LIN {X -277.944,Y 0.000,Z 80.000,A 0.000,B 0.000,C 180.000,E1 0.000} C_DIS
LIN {X -277.576,Y -14.309,Z 80.000,A 0.000,B 0.000,C 180.000,E1 0.000} C_DIS
LIN {X -276.472,Y -28.580,Z 80.000,A 0.000,B 0.000,C 180.000,E1 0.000} C_DIS
LIN {X -274.635,Y -42.773,Z 80.000,A 0.000,B 0.000,C 180.000,E1 0.000} C_DIS
LIN {X -272.067,Y -56.854,Z 80.000,A 0.000,B 0.000,C 180.000,E1 0.000} C_DIS
LIN {X -268.780,Y -70.785,Z 80.000,A 0.000,B 0.000,C 180.000,E1 0.000} C_DIS
LIN {X -264.780,Y -84.527,Z 80.000,A 0.000,B 0.000,C 180.000,E1 0.000} C_DIS
LIN {X -260.078,Y -98.045,Z 80.000,A 0.000,B 0.000,C 180.000,E1 0.000} C_DIS
LIN {X -254.685,Y -111.305,Z 80.000,A 0.000,B 0.000,C 180.000,E1 0.000} C_DIS
LIN {X -248.618,Y -124.267,Z 80.000,A 0.000,B 0.000,C 180.000,E1 0.000} C_DIS
LIN {X -241.892,Y -136.901,Z 80.000,A 0.000,B 0.000,C 180.000,E1 0.000} C_DIS
LIN {X -234.523,Y -149.172,Z 80.000,A 0.000,B 0.000,C 180.000,E1 0.000} C_DIS
LIN {X -226.533,Y -161.047,Z 80.000,A 0.000,B 0.000,C 180.000,E1 0.000} C_DIS
LIN {X -217.943,Y -172.495,Z 80.000,A 0.000,B 0.000,C 180.000,E1 0.000} C_DIS
LIN {X -208.773,Y -183.486,Z 80.000,A 0.000,B 0.000,C 180.000,E1 0.000} C_DIS
LIN {X -199.051,Y -193.990,Z 80.000,A 0.000,B 0.000,C 180.000,E1 0.000} C_DIS
LIN {X -188.801,Y -203.979,Z 80.000,A 0.000,B 0.000,C 180.000,E1 0.000} C_DIS
LIN {X -178.050,Y -213.428,Z 80.000,A 0.000,B 0.000,C 180.000,E1 0.000} C_DIS
LIN {X -166.826,Y -222.311,Z 80.000,A 0.000,B 0.000,C 180.000,E1 0.000} C_DIS
LIN {X -155.161,Y -230.604,Z 80.000,A 0.000,B 0.000,C 180.000,E1 0.000} C_DIS
LIN {X -143.084,Y -238.286,Z 80.000,A 0.000,B 0.000,C 180.000,E1 0.000} C_DIS
LIN {X -130.627,Y -245.336,Z 80.000,A 0.000,B 0.000,C 180.000,E1 0.000} C_DIS
LIN {X -117.825,Y -251.735,Z 80.000,A 0.000,B 0.000,C 180.000,E1 0.000} C_DIS
LIN {X -104.709,Y -257.467,Z 80.000,A 0.000,B 0.000,C 180.000,E1 0.000} C_DIS
LIN {X -91.317,Y -262.516,Z 80.000,A 0.000,B 0.000,C 180.000,E1 0.000} C_DIS
LIN {X -77.682,Y -266.869,Z 80.000,A 0.000,B 0.000,C 180.000,E1 0.000} C_DIS
LIN {X -63.841,Y -270.513,Z 80.000,A 0.000,B 0.000,C 180.000,E1 0.000} C_DIS
LIN {X -49.830,Y -273.441,Z 80.000,A 0.000,B 0.000,C 180.000,E1 0.000} C_DIS
LIN {X -35.687,Y -275.644,Z 80.000,A 0.000,B 0.000,C 180.000,E1 0.000} C_DIS
LIN {X -21.451,Y -277.115,Z 80.000,A 0.000,B 0.000,C 180.000,E1 0.000} C_DIS
LIN {X -7.156,Y -277.853,Z 80.000,A 0.000,B 0.000,C 180.000,E1 0.000} C_DIS
LIN {X 7.156,Y -277.853,Z 80.000,A 0.000,B 0.000,C 180.000,E1 0.000} C_DIS
LIN {X 21.451,Y -277.115,Z 80.000,A 0.000,B 0.000,C 180.000,E1 0.000} C_DIS
LIN {X 35.687,Y -275.644,Z 80.000,A 0.000,B 0.000,C 180.000,E1 0.000} C_DIS
LIN {X 49.830,Y -273.441,Z 80.000,A 0.000,B 0.000,C 180.000,E1 0.000} C_DIS
LIN {X 63.841,Y -270.513,Z 80.000,A 0.000,B 0.000,C 180.000,E1 0.000} C_DIS
LIN {X 77.682,Y -266.869,Z 80.000,A 0.000,B 0.000,C 180.000,E1 0.000} C_DIS
LIN {X 91.317,Y -262.516,Z 80.000,A 0.000,B 0.000,C 180.000,E1 0.000} C_DIS
LIN {X 104.709,Y -257.467,Z 80.000,A 0.000,B 0.000,C 180.000,E1 0.000} C_DIS
LIN {X 117.825,Y -251.735,Z 80.000,A 0.000,B 0.000,C 180.000,E1 0.000} C_DIS
LIN {X 130.627,Y -245.336,Z 80.000,A 0.000,B 0.000,C 180.000,E1 0.000} C_DIS
LIN {X 143.084,Y -238.286,Z 80.000,A 0.000,B 0.000,C 180.000,E1 0.000} C_DIS
LIN {X 155.161,Y -230.604,Z 80.000,A 0.000,B 0.000,C 180.000,E1 0.000} C_DIS
LIN {X 166.826,Y -222.311,Z 80.000,A 0.000,B 0.000,C 180.000,E1 0.000} C_DIS
LIN {X 178.050,Y -213.428,Z 80.000,A 0.000,B 0.000,C 180.000,E1 0.000} C_DIS
LIN {X 188.801,Y -203.979,Z 80.000,A 0.000,B 0.000,C 180.000,E1 0.000} C_DIS
LIN {X 199.051,Y -193.990,Z 80.000,A 0.000,B 0.000,C 180.000,E1 0.000} C_DIS
LIN {X 208.773,Y -183.486,Z 80.000,A 0.000,B 0.000,C 180.000,E1 0.000} C_DIS
LIN {X 217.943,Y -172.495,Z 80.000,A 0.000,B 0.000,C 180.000,E1 0.000} C_DIS
LIN {X 226.533,Y -161.047,Z 80.000,A 0.000,B 0.000,C 180.000,E1 0.000} C_DIS
LIN {X 234.523,Y -149.172,Z 80.000,A 0.000,B 0.000,C 180.000,E1 0.000} C_DIS
LIN {X 241.892,Y -136.901,Z 80.000,A 0.000,B 0.000,C 180.000,E1 0.000} C_DIS
LIN {X 248.618,Y -124.268,Z 80.000,A 0.000,B 0.000,C 180.000,E1 0.000} C_DIS
LIN {X 254.686,Y -111.304,Z 80.000,A 0.000,B 0.000,C 180.000,E1 0.000} C_DIS
LIN {X 260.078,Y -98.045,Z 80.000,A 0.000,B 0.000,C 180.000,E1 0.000} C_DIS
LIN {X 264.780,Y -84.527,Z 80.000,A 0.000,B 0.000,C 180.000,E1 0.000} C_DIS
LIN {X 268.780,Y -70.785,Z 80.000,A 0.000,B 0.000,C 180.000,E1 0.000} C_DIS
LIN {X 272.067,Y -56.854,Z 80.000,A 0.000,B 0.000,C 180.000,E1 0.000} C_DIS
LIN {X 274.635,Y -42.773,Z 80.000,A 0.000,B 0.000,C 180.000,E1 0.000} C_DIS
LIN {X 276.472,Y -28.580,Z 80.000,A 0.000,B 0.000,C 180.000,E1 0.000} C_DIS
LIN {X 277.576,Y -14.309,Z 80.000,A 0.000,B 0.000,C 180.000,E1 0.000} C_DIS
LIN {X 277.944,Y 0.000,Z 80.000,A 0.000,B 0.000,C 180.000,E1 0.000} C_DIS
LIN {X 277.576,Y 14.309,Z 80.000,A 0.000,B 0.000,C 180.000,E1 0.000} C_DIS
LIN {X 276.472,Y 28.580,Z 80.000,A 0.000,B 0.000,C 180.000,E1 0.000} C_DIS
LIN {X 274.635,Y 42.773,Z 80.000,A 0.000,B 0.000,C 180.000,E1 0.000} C_DIS
LIN {X 272.067,Y 56.854,Z 80.000,A 0.000,B 0.000,C 180.000,E1 0.000} C_DIS
LIN {X 268.780,Y 70.785,Z 80.000,A 0.000,B 0.000,C 180.000,E1 0.000} C_DIS
LIN {X 264.780,Y 84.527,Z 80.000,A 0.000,B 0.000,C 180.000,E1 0.000} C_DIS
LIN {X 260.078,Y 98.045,Z 80.000,A 0.000,B 0.000,C 180.000,E1 0.000} C_DIS
LIN {X 254.685,Y 111.305,Z 80.000,A 0.000,B 0.000,C 180.000,E1 0.000} C_DIS
LIN {X 252.753,Y 115.434,Z 80.000,A 0.000,B 0.000,C 180.000,E1 0.000} C_DIS
LIN {X 248.618,Y 124.267,Z 80.000,A 0.000,B 0.000,C 180.000,E1 0.000} C_DIS
LIN {X 241.892,Y 136.901,Z 80.000,A 0.000,B 0.000,C 180.000,E1 0.000} C_DIS
LIN {X 234.523,Y 149.172,Z 80.000,A 0.000,B 0.000,C 180.000,E1 0.000} C_DIS
LIN {X 226.533,Y 161.047,Z 80.000,A 0.000,B 0.000,C 180.000,E1 0.000} C_DIS
LIN {X 217.943,Y 172.495,Z 80.000,A 0.000,B 0.000,C 180.000,E1 0.000} C_DIS
LIN {X 208.773,Y 183.486,Z 80.000,A 0.000,B 0.000,C 180.000,E1 0.000} C_DIS
LIN {X 199.051,Y 193.990,Z 80.000,A 0.000,B 0.000,C 180.000,E1 0.000} C_DIS
LIN {X 188.801,Y 203.979,Z 80.000,A 0.000,B 0.000,C 180.000,E1 0.000} C_DIS
LIN {X 178.050,Y 213.428,Z 80.000,A 0.000,B 0.000,C 180.000,E1 0.000} C_DIS
LIN {X 166.826,Y 222.311,Z 80.000,A 0.000,B 0.000,C 180.000,E1 0.000} C_DIS
LIN {X 155.161,Y 230.604,Z 80.000,A 0.000,B 0.000,C 180.000,E1 0.000} C_DIS
LIN {X 143.084,Y 238.286,Z 80.000,A 0.000,B 0.000,C 180.000,E1 0.000} C_DIS
LIN {X 130.627,Y 245.336,Z 80.000,A 0.000,B 0.000,C 180.000,E1 0.000} C_DIS
LIN {X 117.825,Y 251.735,Z 80.000,A 0.000,B 0.000,C 180.000,E1 0.000} C_DIS
LIN {X 104.709,Y 257.467,Z 80.000,A 0.000,B 0.000,C 180.000,E1 0.000} C_DIS
LIN {X 91.317,Y 262.516,Z 80.000,A 0.000,B 0.000,C 180.000,E1 0.000} C_DIS
LIN {X 77.682,Y 266.869,Z 80.000,A 0.000,B 0.000,C 180.000,E1 0.000} C_DIS
;rapid-leaky
$VEL.CP=0.3
LIN {X 73.337,Y 251.943,Z 80.000,A 0.000,B 0.000,C 180.000,E1 0.000} C_DIS
;bead-perimeter_inner
$VEL.CP=0.73
LIN {X 60.270,Y 255.384,Z 80.000,A 0.000,B 0.000,C 180.000,E1 0.000} C_DIS
LIN {X 47.043,Y 258.148,Z 80.000,A 0.000,B 0.000,C 180.000,E1 0.000} C_DIS
LIN {X 33.691,Y 260.228,Z 80.000,A 0.000,B 0.000,C 180.000,E1 0.000} C_DIS
LIN {X 20.251,Y 261.617,Z 80.000,A 0.000,B 0.000,C 180.000,E1 0.000} C_DIS
LIN {X 6.755,Y 262.313,Z 80.000,A 0.000,B 0.000,C 180.000,E1 0.000} C_DIS
LIN {X -6.755,Y 262.313,Z 80.000,A 0.000,B 0.000,C 180.000,E1 0.000} C_DIS
LIN {X -20.251,Y 261.617,Z 80.000,A 0.000,B 0.000,C 180.000,E1 0.000} C_DIS
LIN {X -33.691,Y 260.228,Z 80.000,A 0.000,B 0.000,C 180.000,E1 0.000} C_DIS
LIN {X -47.043,Y 258.148,Z 80.000,A 0.000,B 0.000,C 180.000,E1 0.000} C_DIS
LIN {X -60.270,Y 255.384,Z 80.000,A 0.000,B 0.000,C 180.000,E1 0.000} C_DIS
LIN {X -73.337,Y 251.943,Z 80.000,A 0.000,B 0.000,C 180.000,E1 0.000} C_DIS
LIN {X -86.210,Y 247.833,Z 80.000,A 0.000,B 0.000,C 180.000,E1 0.000} C_DIS
LIN {X -98.853,Y 243.067,Z 80.000,A 0.000,B 0.000,C 180.000,E1 0.000} C_DIS
LIN {X -111.235,Y 237.656,Z 80.000,A 0.000,B 0.000,C 180.000,E1 0.000} C_DIS
LIN {X -123.321,Y 231.615,Z 80.000,A 0.000,B 0.000,C 180.000,E1 0.000} C_DIS
LIN {X -135.081,Y 224.959,Z 80.000,A 0.000,B 0.000,C 180.000,E1 0.000} C_DIS
LIN {X -146.484,Y 217.706,Z 80.000,A 0.000,B 0.000,C 180.000,E1 0.000} C_DIS
LIN {X -157.496,Y 209.877,Z 80.000,A 0.000,B 0.000,C 180.000,E1 0.000} C_DIS
LIN {X -168.092,Y 201.491,Z 80.000,A 0.000,B 0.000,C 180.000,E1 0.000} C_DIS
LIN {X -178.242,Y 192.570,Z 80.000,A 0.000,B 0.000,C 180.000,E1 0.000} C_DIS
LIN {X -187.918,Y 183.141,Z 80.000,A 0.000,B 0.000,C 180.000,E1 0.000} C_DIS
LIN {X -197.096,Y 173.224,Z 80.000,A 0.000,B 0.000,C 180.000,E1 0.000} C_DIS
LIN {X -205.754,Y 162.847,Z 80.000,A 0.000,B 0.000,C 180.000,E1 0.000} C_DIS
LIN {X -213.863,Y 152.040,Z 80.000,A 0.000,B 0.000,C 180.000,E1 0.000} C_DIS
LIN {X -221.406,Y 140.829,Z 80.000,A 0.000,B 0.000,C 180.000,E1 0.000} C_DIS
LIN {X -228.363,Y 129.244,Z 80.000,A 0.000,B 0.000,C 180.000,E1 0.000} C_DIS
LIN {X -234.713,Y 117.317,Z 80.000,A 0.000,B 0.000,C 180.000,E1 0.000} C_DIS
LIN {X -240.441,Y 105.079,Z 80.000,A 0.000,B 0.000,C 180.000,E1 0.000} C_DIS
LIN {X -245.532,Y 92.562,Z 80.000,A 0.000,B 0.000,C 180.000,E1 0.000} C_DIS
LIN {X -249.971,Y 79.800,Z 80.000,A 0.000,B 0.000,C 180.000,E1 0.000} C_DIS
LIN {X -253.748,Y 66.826,Z 80.000,A 0.000,B 0.000,C 180.000,E1 0.000} C_DIS
LIN {X -256.851,Y 53.674,Z 80.000,A 0.000,B 0.000,C 180.000,E1 0.000} C_DIS
LIN {X -259.275,Y 40.380,Z 80.000,A 0.000,B 0.000,C 180.000,E1 0.000} C_DIS
LIN {X -261.009,Y 26.982,Z 80.000,A 0.000,B 0.000,C 180.000,E1 0.000} C_DIS
LIN {X -262.051,Y 13.509,Z 80.000,A 0.000,B 0.000,C 180.000,E1 0.000} C_DIS
LIN {X -262.399,Y 0.000,Z 80.000,A 0.000,B 0.000,C 180.000,E1 0.000} C_DIS
LIN {X -262.051,Y -13.509,Z 80.000,A 0.000,B 0.000,C 180.000,E1 0.000} C_DIS
LIN {X -261.009,Y -26.982,Z 80.000,A 0.000,B 0.000,C 180.000,E1 0.000} C_DIS
LIN {X -259.275,Y -40.380,Z 80.000,A 0.000,B 0.000,C 180.000,E1 0.000} C_DIS
LIN {X -256.851,Y -53.674,Z 80.000,A 0.000,B 0.000,C 180.000,E1 0.000} C_DIS
LIN {X -253.748,Y -66.826,Z 80.000,A 0.000,B 0.000,C 180.000,E1 0.000} C_DIS
LIN {X -249.971,Y -79.800,Z 80.000,A 0.000,B 0.000,C 180.000,E1 0.000} C_DIS
LIN {X -245.532,Y -92.562,Z 80.000,A 0.000,B 0.000,C 180.000,E1 0.000} C_DIS
LIN {X -240.441,Y -105.080,Z 80.000,A 0.000,B 0.000,C 180.000,E1 0.000} C_DIS
LIN {X -234.713,Y -117.317,Z 80.000,A 0.000,B 0.000,C 180.000,E1 0.000} C_DIS
LIN {X -228.363,Y -129.244,Z 80.000,A 0.000,B 0.000,C 180.000,E1 0.000} C_DIS
LIN {X -221.406,Y -140.829,Z 80.000,A 0.000,B 0.000,C 180.000,E1 0.000} C_DIS
LIN {X -213.863,Y -152.040,Z 80.000,A 0.000,B 0.000,C 180.000,E1 0.000} C_DIS
LIN {X -205.754,Y -162.847,Z 80.000,A 0.000,B 0.000,C 180.000,E1 0.000} C_DIS
LIN {X -197.096,Y -173.224,Z 80.000,A 0.000,B 0.000,C 180.000,E1 0.000} C_DIS
LIN {X -187.918,Y -183.141,Z 80.000,A 0.000,B 0.000,C 180.000,E1 0.000} C_DIS
LIN {X -178.242,Y -192.570,Z 80.000,A 0.000,B 0.000,C 180.000,E1 0.000} C_DIS
LIN {X -168.092,Y -201.491,Z 80.000,A 0.000,B 0.000,C 180.000,E1 0.000} C_DIS
LIN {X -157.496,Y -209.877,Z 80.000,A 0.000,B 0.000,C 180.000,E1 0.000} C_DIS
LIN {X -146.484,Y -217.706,Z 80.000,A 0.000,B 0.000,C 180.000,E1 0.000} C_DIS
LIN {X -135.081,Y -224.959,Z 80.000,A 0.000,B 0.000,C 180.000,E1 0.000} C_DIS
LIN {X -123.321,Y -231.615,Z 80.000,A 0.000,B 0.000,C 180.000,E1 0.000} C_DIS
LIN {X -111.235,Y -237.656,Z 80.000,A 0.000,B 0.000,C 180.000,E1 0.000} C_DIS
LIN {X -98.853,Y -243.067,Z 80.000,A 0.000,B 0.000,C 180.000,E1 0.000} C_DIS
LIN {X -86.210,Y -247.833,Z 80.000,A 0.000,B 0.000,C 180.000,E1 0.000} C_DIS
LIN {X -73.337,Y -251.943,Z 80.000,A 0.000,B 0.000,C 180.000,E1 0.000} C_DIS
LIN {X -60.270,Y -255.384,Z 80.000,A 0.000,B 0.000,C 180.000,E1 0.000} C_DIS
LIN {X -47.043,Y -258.148,Z 80.000,A 0.000,B 0.000,C 180.000,E1 0.000} C_DIS
LIN {X -33.691,Y -260.228,Z 80.000,A 0.000,B 0.000,C 180.000,E1 0.000} C_DIS
LIN {X -20.251,Y -261.617,Z 80.000,A 0.000,B 0.000,C 180.000,E1 0.000} C_DIS
LIN {X -6.755,Y -262.313,Z 80.000,A 0.000,B 0.000,C 180.000,E1 0.000} C_DIS
LIN {X 6.755,Y -262.313,Z 80.000,A 0.000,B 0.000,C 180.000,E1 0.000} C_DIS
LIN {X 20.251,Y -261.617,Z 80.000,A 0.000,B 0.000,C 180.000,E1 0.000} C_DIS
LIN {X 33.691,Y -260.228,Z 80.000,A 0.000,B 0.000,C 180.000,E1 0.000} C_DIS
LIN {X 47.043,Y -258.148,Z 80.000,A 0.000,B 0.000,C 180.000,E1 0.000} C_DIS
LIN {X 60.270,Y -255.384,Z 80.000,A 0.000,B 0.000,C 180.000,E1 0.000} C_DIS
LIN {X 73.337,Y -251.943,Z 80.000,A 0.000,B 0.000,C 180.000,E1 0.000} C_DIS
LIN {X 86.210,Y -247.833,Z 80.000,A 0.000,B 0.000,C 180.000,E1 0.000} C_DIS
LIN {X 98.853,Y -243.067,Z 80.000,A 0.000,B 0.000,C 180.000,E1 0.000} C_DIS
LIN {X 111.235,Y -237.656,Z 80.000,A 0.000,B 0.000,C 180.000,E1 0.000} C_DIS
LIN {X 123.321,Y -231.615,Z 80.000,A 0.000,B 0.000,C 180.000,E1 0.000} C_DIS
LIN {X 135.081,Y -224.959,Z 80.000,A 0.000,B 0.000,C 180.000,E1 0.000} C_DIS
LIN {X 146.484,Y -217.706,Z 80.000,A 0.000,B 0.000,C 180.000,E1 0.000} C_DIS
LIN {X 157.496,Y -209.877,Z 80.000,A 0.000,B 0.000,C 180.000,E1 0.000} C_DIS
LIN {X 168.092,Y -201.491,Z 80.000,A 0.000,B 0.000,C 180.000,E1 0.000} C_DIS
LIN {X 178.242,Y -192.570,Z 80.000,A 0.000,B 0.000,C 180.000,E1 0.000} C_DIS
LIN {X 187.918,Y -183.141,Z 80.000,A 0.000,B 0.000,C 180.000,E1 0.000} C_DIS
LIN {X 197.096,Y -173.224,Z 80.000,A 0.000,B 0.000,C 180.000,E1 0.000} C_DIS
LIN {X 205.754,Y -162.847,Z 80.000,A 0.000,B 0.000,C 180.000,E1 0.000} C_DIS
LIN {X 213.863,Y -152.040,Z 80.000,A 0.000,B 0.000,C 180.000,E1 0.000} C_DIS
LIN {X 221.406,Y -140.829,Z 80.000,A 0.000,B 0.000,C 180.000,E1 0.000} C_DIS
LIN {X 228.363,Y -129.244,Z 80.000,A 0.000,B 0.000,C 180.000,E1 0.000} C_DIS
LIN {X 234.713,Y -117.317,Z 80.000,A 0.000,B 0.000,C 180.000,E1 0.000} C_DIS
LIN {X 240.441,Y -105.079,Z 80.000,A 0.000,B 0.000,C 180.000,E1 0.000} C_DIS
LIN {X 245.532,Y -92.562,Z 80.000,A 0.000,B 0.000,C 180.000,E1 0.000} C_DIS
LIN {X 249.971,Y -79.800,Z 80.000,A 0.000,B 0.000,C 180.000,E1 0.000} C_DIS
LIN {X 253.748,Y -66.826,Z 80.000,A 0.000,B 0.000,C 180.000,E1 0.000} C_DIS
LIN {X 256.851,Y -53.674,Z 80.000,A 0.000,B 0.000,C 180.000,E1 0.000} C_DIS
LIN {X 259.275,Y -40.380,Z 80.000,A 0.000,B 0.000,C 180.000,E1 0.000} C_DIS
LIN {X 261.009,Y -26.982,Z 80.000,A 0.000,B 0.000,C 180.000,E1 0.000} C_DIS
LIN {X 262.051,Y -13.509,Z 80.000,A 0.000,B 0.000,C 180.000,E1 0.000} C_DIS
LIN {X 262.399,Y 0.000,Z 80.000,A 0.000,B 0.000,C 180.000,E1 0.000} C_DIS
LIN {X 262.051,Y 13.509,Z 80.000,A 0.000,B 0.000,C 180.000,E1 0.000} C_DIS
LIN {X 261.009,Y 26.982,Z 80.000,A 0.000,B 0.000,C 180.000,E1 0.000} C_DIS
LIN {X 259.275,Y 40.380,Z 80.000,A 0.000,B 0.000,C 180.000,E1 0.000} C_DIS
LIN {X 256.851,Y 53.674,Z 80.000,A 0.000,B 0.000,C 180.000,E1 0.000} C_DIS
LIN {X 253.748,Y 66.826,Z 80.000,A 0.000,B 0.000,C 180.000,E1 0.000} C_DIS
LIN {X 249.971,Y 79.800,Z 80.000,A 0.000,B 0.000,C 180.000,E1 0.000} C_DIS
LIN {X 245.532,Y 92.562,Z 80.000,A 0.000,B 0.000,C 180.000,E1 0.000} C_DIS
LIN {X 240.441,Y 105.080,Z 80.000,A 0.000,B 0.000,C 180.000,E1 0.000} C_DIS
LIN {X 238.678,Y 108.847,Z 80.000,A 0.000,B 0.000,C 180.000,E1 0.000} C_DIS
LIN {X 234.713,Y 117.317,Z 80.000,A 0.000,B 0.000,C 180.000,E1 0.000} C_DIS
LIN {X 228.363,Y 129.244,Z 80.000,A 0.000,B 0.000,C 180.000,E1 0.000} C_DIS
LIN {X 221.406,Y 140.829,Z 80.000,A 0.000,B 0.000,C 180.000,E1 0.000} C_DIS
LIN {X 213.863,Y 152.040,Z 80.000,A 0.000,B 0.000,C 180.000,E1 0.000} C_DIS
LIN {X 205.754,Y 162.847,Z 80.000,A 0.000,B 0.000,C 180.000,E1 0.000} C_DIS
LIN {X 197.096,Y 173.224,Z 80.000,A 0.000,B 0.000,C 180.000,E1 0.000} C_DIS
LIN {X 187.918,Y 183.141,Z 80.000,A 0.000,B 0.000,C 180.000,E1 0.000} C_DIS
LIN {X 178.242,Y 192.570,Z 80.000,A 0.000,B 0.000,C 180.000,E1 0.000} C_DIS
LIN {X 168.092,Y 201.491,Z 80.000,A 0.000,B 0.000,C 180.000,E1 0.000} C_DIS
LIN {X 157.496,Y 209.877,Z 80.000,A 0.000,B 0.000,C 180.000,E1 0.000} C_DIS
LIN {X 146.484,Y 217.706,Z 80.000,A 0.000,B 0.000,C 180.000,E1 0.000} C_DIS
LIN {X 135.081,Y 224.959,Z 80.000,A 0.000,B 0.000,C 180.000,E1 0.000} C_DIS
LIN {X 123.321,Y 231.615,Z 80.000,A 0.000,B 0.000,C 180.000,E1 0.000} C_DIS
LIN {X 111.235,Y 237.656,Z 80.000,A 0.000,B 0.000,C 180.000,E1 0.000} C_DIS
LIN {X 98.853,Y 243.067,Z 80.000,A 0.000,B 0.000,C 180.000,E1 0.000} C_DIS
LIN {X 86.210,Y 247.833,Z 80.000,A 0.000,B 0.000,C 180.000,E1 0.000} C_DIS
LIN {X 73.337,Y 251.943,Z 80.000,A 0.000,B 0.000,C 180.000,E1 0.000} C_DIS
;rapid-leaky
$VEL.CP=0.3
LIN {X -163.493,Y 181.889,Z 80.000,A 0.000,B 0.000,C 180.000,E1 0.000} C_DIS
;bead-sparse_infill
$VEL.CP=0.73
LIN {X -182.087,Y 163.294,Z 80.000,A 0.000,B 0.000,C 180.000,E1 0.000} C_DIS
LIN {X -183.751,Y 161.496,Z 80.000,A 0.000,B 0.000,C 180.000,E1 0.000} C_DIS
LIN {X -191.823,Y 151.821,Z 80.000,A 0.000,B 0.000,C 180.000,E1 0.000} C_DIS
LIN {X -199.383,Y 141.747,Z 80.000,A 0.000,B 0.000,C 180.000,E1 0.000} C_DIS
LIN {X -206.416,Y 131.294,Z 80.000,A 0.000,B 0.000,C 180.000,E1 0.000} C_DIS
LIN {X -212.902,Y 120.493,Z 80.000,A 0.000,B 0.000,C 180.000,E1 0.000} C_DIS
LIN {X -218.822,Y 109.374,Z 80.000,A 0.000,B 0.000,C 180.000,E1 0.000} C_DIS
LIN {X -224.162,Y 97.965,Z 80.000,A 0.000,B 0.000,C 180.000,E1 0.000} C_DIS
LIN {X -228.908,Y 86.295,Z 80.000,A 0.000,B 0.000,C 180.000,E1 0.000} C_DIS
LIN {X -233.047,Y 74.397,Z 80.000,A 0.000,B 0.000,C 180.000,E1 0.000} C_DIS
LIN {X -236.567,Y 62.302,Z 80.000,A 0.000,B 0.000,C 180.000,E1 0.000} C_DIS
LIN {X -239.461,Y 50.040,Z 80.000,A 0.000,B 0.000,C 180.000,E1 0.000} C_DIS
LIN {X -241.721,Y 37.645,Z 80.000,A 0.000,B 0.000,C 180.000,E1 0.000} C_DIS
LIN {X -243.338,Y 25.156,Z 80.000,A 0.000,B 0.000,C 180.000,E1 0.000} C_DIS
LIN {X -244.309,Y 12.595,Z 80.000,A 0.000,B 0.000,C 180.000,E1 0.000} C_DIS
LIN {X -244.633,Y 0.000,Z 80.000,A 0.000,B 0.000,C 180.000,E1 0.000} C_DIS
LIN {X -244.309,Y -12.595,Z 80.000,A 0.000,B 0.000,C 180.000,E1 0.000} C_DIS
LIN {X -243.338,Y -25.156,Z 80.000,A 0.000,B 0.000,C 180.000,E1 0.000} C_DIS
LIN {X -241.721,Y -37.645,Z 80.000,A 0.000,B 0.000,C 180.000,E1 0.000} C_DIS
LIN {X -239.461,Y -50.040,Z 80.000,A 0.000,B 0.000,C 180.000,E1 0.000} C_DIS
LIN {X -239.266,Y -50.863,Z 80.000,A 0.000,B 0.000,C 180.000,E1 0.000} C_DIS
LIN {X 50.813,Y 239.216,Z 80.000,A 0.000,B 0.000,C 180.000,E1 0.000} C_DIS
LIN {X 56.190,Y 238.093,Z 80.000,A 0.000,B 0.000,C 180.000,E1 0.000} C_DIS
LIN {X 68.372,Y 234.885,Z 80.000,A 0.000,B 0.000,C 180.000,E1 0.000} C_DIS
LIN {X 80.373,Y 231.054,Z 80.000,A 0.000,B 0.000,C 180.000,E1 0.000} C_DIS
LIN {X 92.160,Y 226.610,Z 80.000,A 0.000,B 0.000,C 180.000,E1 0.000} C_DIS
LIN {X 103.704,Y 221.566,Z 80.000,A 0.000,B 0.000,C 180.000,E1 0.000} C_DIS
LIN {X 114.971,Y 215.934,Z 80.000,A 0.000,B 0.000,C 180.000,E1 0.000} C_DIS
LIN {X 125.935,Y 209.728,Z 80.000,A 0.000,B 0.000,C 180.000,E1 0.000} C_DIS
LIN {X 136.566,Y 202.966,Z 80.000,A 0.000,B 0.000,C 180.000,E1 0.000} C_DIS
LIN {X 146.833,Y 195.667,Z 80.000,A 0.000,B 0.000,C 180.000,E1 0.000} C_DIS
LIN {X 156.550,Y 187.976,Z 80.000,A 0.000,B 0.000,C 180.000,E1 0.000} C_DIS
LIN {X -187.922,Y -156.497,Z 80.000,A 0.000,B 0.000,C 180.000,E1 0.000} C_DIS
LIN {X -183.751,Y -161.496,Z 80.000,A 0.000,B 0.000,C 180.000,E1 0.000} C_DIS
LIN {X -175.195,Y -170.741,Z 80.000,A 0.000,B 0.000,C 180.000,E1 0.000} C_DIS
LIN {X -166.174,Y -179.532,Z 80.000,A 0.000,B 0.000,C 180.000,E1 0.000} C_DIS
LIN {X -156.711,Y -187.849,Z 80.000,A 0.000,B 0.000,C 180.000,E1 0.000} C_DIS
LIN {X -146.833,Y -195.667,Z 80.000,A 0.000,B 0.000,C 180.000,E1 0.000} C_DIS
LIN {X -136.566,Y -202.966,Z 80.000,A 0.000,B 0.000,C 180.000,E1 0.000} C_DIS
LIN {X -125.935,Y -209.728,Z 80.000,A 0.000,B 0.000,C 180.000,E1 0.000} C_DIS
LIN {X -114.971,Y -215.934,Z 80.000,A 0.000,B 0.000,C 180.000,E1 0.000} C_DIS
LIN {X -103.704,Y -221.566,Z 80.000,A 0.000,B 0.000,C 180.000,E1 0.000} C_DIS
LIN {X -98.352,Y -223.904,Z 80.000,A 0.000,B 0.000,C 180.000,E1 0.000} C_DIS
LIN {X 223.956,Y 98.405,Z 80.000,A 0.000,B 0.000,C 180.000,E1 0.000} C_DIS
LIN {X 224.162,Y 97.966,Z 80.000,A 0.000,B 0.000,C 180.000,E1 0.000} C_DIS
LIN {X 228.908,Y 86.295,Z 80.000,A 0.000,B 0.000,C 180.000,E1 0.000} C_DIS
LIN {X 233.047,Y 74.397,Z 80.000,A 0.000,B 0.000,C 180.000,E1 0.000} C_DIS
LIN {X 236.567,Y 62.302,Z 80.000,A 0.000,B 0.000,C 180.000,E1 0.000} C_DIS
LIN {X 239.461,Y 50.040,Z 80.000,A 0.000,B 0.000,C 180.000,E1 0.000} C_DIS
LIN {X 241.721,Y 37.645,Z 80.000,A 0.000,B 0.000,C 180.000,E1 0.000} C_DIS
LIN {X 243.338,Y 25.156,Z 80.000,A 0.000,B 0.000,C 180.000,E1 0.000} C_DIS
LIN {X 244.309,Y 12.595,Z 80.000,A 0.000,B 0.000,C 180.000,E1 0.000} C_DIS
LIN {X 244.633,Y 0.000,Z 80.000,A 0.000,B 0.000,C 180.000,E1 0.000} C_DIS
LIN {X 244.309,Y -12.595,Z 80.000,A 0.000,B 0.000,C 180.000,E1 0.000} C_DIS
LIN {X 243.338,Y -25.156,Z 80.000,A 0.000,B 0.000,C 180.000,E1 0.000} C_DIS
LIN {X 241.721,Y -37.645,Z 80.000,A 0.000,B 0.000,C 180.000,E1 0.000} C_DIS
LIN {X 241.015,Y -41.514,Z 80.000,A 0.000,B 0.000,C 180.000,E1 0.000} C_DIS
LIN {X 41.491,Y -241.039,Z 80.000,A 0.000,B 0.000,C 180.000,E1 0.000} C_DIS
;rapid-leaky
$VEL.CP=0.3
LIN {X -176.208,Y 211.220,Z 90.000,A 0.000,B 0.000,C 180.000,E1 0.000} C_DIS
;bead-perimeter_outer
$VEL.CP=0.69
LIN {X -186.848,Y 201.870,Z 90.000,A 0.000,B 0.000,C 180.000,E1 0.000} C_DIS
LIN {X -197.001,Y 191.974,Z 90.000,A 0.000,B 0.000,C 180.000,E1 0.000} C_DIS
LIN {X -206.613,Y 181.588,Z 90.000,A 0.000,B 0.000,C 180.000,E1 0.000} C_DIS
LIN {X -215.687,Y 170.711,Z 90.000,A 0.000,B 0.000,C 180.000,E1 0.000} C_DIS
LIN {X -224.189,Y 159.381,Z 90.000,A 0.000,B 0.000,C 180.000,E1 0.000} C_DIS
LIN {X -232.097,Y 147.628,Z 90.000,A 0.000,B 0.000,C 180.000,E1 0.000} C_DIS
LIN {X -239.390,Y 135.485,Z 90.000,A 0.000,B 0.000,C 180.000,E1 0.000} C_DIS
LIN {X -246.047,Y 122.982,Z 90.000,A 0.000,B 0.000,C 180.000,E1 0.000} C_DIS
LIN {X -252.050,Y 110.154,Z 90.000,A 0.000,B 0.000,C 180.000,E1 0.000} C_DIS
LIN {X -257.387,Y 97.031,Z 90.000,A 0.000,B 0.000,C 180.000,E1 0.000} C_DIS
LIN {X -262.041,Y 83.652,Z 90.000,A 0.000,B 0.000,C 180.000,E1 0.000} C_DIS
LIN {X -266.000,Y 70.053,Z 90.000,A 0.000,B 0.000,C 180.000,E1 0.000} C_DIS
LIN {X -269.253,Y 56.266,Z 90.000,A 0.000,B 0.000,C 180.000,E1 0.000} C_DIS
LIN {X -271.794,Y 42.330,Z 90.000,A 0.000,B 0.000,C 180.000,E1 0.000} C_DIS
LIN {X -273.612,Y 28.283,Z 90.000,A 0.000,B 0.000,C 180.000,E1 0.000} C_DIS
LIN {X -274.705,Y 14.159,Z 90.000,A 0.000,B 0.000,C 180.000,E1 0.000} C_DIS
LIN {X -275.070,Y 0.000,Z 90.000,A 0.000,B 0.000,C 180.000,E1 0.000} C_DIS
LIN {X -274.705,Y -14.159,Z 90.000,A 0.000,B 0.000,C 180.000,E1 0.000} C_DIS
LIN {X -273.612,Y -28.283,Z 90.000,A 0.000,B 0.000,C 180.000,E1 0.000} C_DIS
LIN {X -271.794,Y -42.330,Z 90.000,A 0.000,B 0.000,C 180.000,E1 0.000} C_DIS
LIN {X -269.253,Y -56.266,Z 90.000,A 0.000,B 0.000,C 180.000,E1 0.000} C_DIS
LIN {X -266.000,Y -70.053,Z 90.000,A 0.000,B 0.000,C 180.000,E1 0.000} C_DIS
LIN {X -262.041,Y -83.652,Z 90.000,A 0.000,B 0.000,C 180.000,E1 0.000} C_DIS
LIN {X -257.387,Y -97.031,Z 90.000,A 0.000,B 0.000,C 180.000,E1 0.000} C_DIS
LIN {X -252.050,Y -110.154,Z 90.000,A 0.000,B 0.000,C 180.000,E1 0.000} C_DIS
LIN {X -246.047,Y -122.982,Z 90.000,A 0.000,B 0.000,C 180.000,E1 0.000} C_DIS
LIN {X -239.390,Y -135.485,Z 90.000,A 0.000,B 0.000,C 180.000,E1 0.000} C_DIS
LIN {X -232.097,Y -147.628,Z 90.000,A 0.000,B 0.000,C 180.000,E1 0.000} C_DIS
LIN {X -224.182,Y -159.392,Z 90.000,A 0.000,B 0.000,C 180.000,E1 0.000} C_DIS
LIN {X -215.687,Y -170.711,Z 90.000,A 0.000,B 0.000,C 180.000,E1 0.000} C_DIS
LIN {X -206.614,Y -181.588,Z 90.000,A 0.000,B 0.000,C 180.000,E1 0.000} C_DIS
LIN {X -196.992,Y -191.983,Z 90.000,A 0.000,B 0.000,C 180.000,E1 0.000} C_DIS
LIN {X -186.848,Y -201.870,Z 90.000,A 0.000,B 0.000,C 180.000,E1 0.000} C_DIS
LIN {X -176.208,Y -211.220,Z 90.000,A 0.000,B 0.000,C 180.000,E1 0.000} C_DIS
LIN {X -165.101,Y -220.011,Z 90.000,A 0.000,B 0.000,C 180.000,E1 0.000} C_DIS
LIN {X -153.556,Y -228.219,Z 90.000,A 0.000,B 0.000,C 180.000,E1 0.000} C_DIS
LIN {X -141.604,Y -235.821,Z 90.000,A 0.000,B 0.000,C 180.000,E1 0.000} C_DIS
LIN {X -129.276,Y -242.799,Z 90.000,A 0.000,B 0.000,C 180.000,E1 0.000} C_DIS
LIN {X -116.606,Y -249.131,Z 90.000,A 0.000,B 0.000,C 180.000,E1 0.000} C_DIS
LIN {X -103.624,Y -254.805,Z 90.000,A 0.000,B 0.000,C 180.000,E1 0.000} C_DIS
LIN {X -90.373,Y -259.801,Z 90.000,A 0.000,B 0.000,C 180.000,E1 0.000} C_DIS
LIN {X -76.878,Y -264.108,Z 90.000,A 0.000,B 0.000,C 180.000,E1 0.000} C_DIS
LIN {X -63.179,Y -267.716,Z 90.000,A 0.000,B 0.000,C 180.000,E1 0.000} C_DIS
LIN {X -49.316,Y -270.613,Z 90.000,A 0.000,B 0.000,C 180.000,E1 0.000} C_DIS
LIN {X -35.318,Y -272.792,Z 90.000,A 0.000,B 0.000,C 180.000,E1 0.000} C_DIS
LIN {X -21.229,Y -274.249,Z 90.000,A 0.000,B 0.000,C 180.000,E1 0.000} C_DIS
LIN {X -7.082,Y -274.979,Z 90.000,A 0.000,B 0.000,C 180.000,E1 0.000} C_DIS
LIN {X 7.082,Y -274.979,Z 90.000,A 0.000,B 0.000,C 180.000,E1 0.000} C_DIS
LIN {X 21.229,Y -274.249,Z 90.000,A 0.000,B 0.000,C 180.000,E1 0.000} C_DIS
LIN {X 35.318,Y -272.792,Z 90.000,A 0.000,B 0.000,C 180.000,E1 0.000} C_DIS
LIN {X 49.316,Y -270.613,Z 90.000,A 0.000,B 0.000,C 180.000,E1 0.000} C_DIS
LIN {X 63.179,Y -267.716,Z 90.000,A 0.000,B 0.000,C 180.000,E1 0.000} C_DIS
LIN {X 76.878,Y -264.108,Z 90.000,A 0.000,B 0.000,C 180.000,E1 0.000} C_DIS
LIN {X 90.373,Y -259.801,Z 90.000,A 0.000,B 0.000,C 180.000,E1 0.000} C_DIS
LIN {X 103.626,Y -254.804,Z 90.000,A 0.000,B 0.000,C 180.000,E1 0.000} C_DIS
LIN {X 116.606,Y -249.131,Z 90.000,A 0.000,B 0.000,C 180.000,E1 0.000} C_DIS
LIN {X 129.276,Y -242.799,Z 90.000,A 0.000,B 0.000,C 180.000,E1 0.000} C_DIS
LIN {X 141.604,Y -235.821,Z 90.000,A 0.000,B 0.000,C 180.000,E1 0.000} C_DIS
LIN {X 153.556,Y -228.219,Z 90.000,A 0.000,B 0.000,C 180.000,E1 0.000} C_DIS
LIN {X 165.101,Y -220.011,Z 90.000,A 0.000,B 0.000,C 180.000,E1 0.000} C_DIS
LIN {X 176.208,Y -211.220,Z 90.000,A 0.000,B 0.000,C 180.000,E1 0.000} C_DIS
LIN {X 186.848,Y -201.870,Z 90.000,A 0.000,B 0.000,C 180.000,E1 0.000} C_DIS
LIN {X 197.001,Y -191.974,Z 90.000,A 0.000,B 0.000,C 180.000,E1 0.000} C_DIS
LIN {X 206.613,Y -181.588,Z 90.000,A 0.000,B 0.000,C 180.000,E1 0.000} C_DIS
LIN {X 215.687,Y -170.711,Z 90.000,A 0.000,B 0.000,C 180.000,E1 0.000} C_DIS
LIN {X 224.189,Y -159.381,Z 90.000,A 0.000,B 0.000,C 180.000,E1 0.000} C_DIS
LIN {X 232.097,Y -147.628,Z 90.000,A 0.000,B 0.000,C 180.000,E1 0.000} C_DIS
LIN {X 239.390,Y -135.485,Z 90.000,A 0.000,B 0.000,C 180.000,E1 0.000} C_DIS
LIN {X 246.047,Y -122.982,Z 90.000,A 0.000,B 0.000,C 180.000,E1 0.000} C_DIS
LIN {X 252.050,Y -110.154,Z 90.000,A 0.000,B 0.000,C 180.000,E1 0.000} C_DIS
LIN {X 257.387,Y -97.031,Z 90.000,A 0.000,B 0.000,C 180.000,E1 0.000} C_DIS
LIN {X 262.041,Y -83.652,Z 90.000,A 0.000,B 0.000,C 180.000,E1 0.000} C_DIS
LIN {X 266.000,Y -70.053,Z 90.000,A 0.000,B 0.000,C 180.000,E1 0.000} C_DIS
LIN {X 269.253,Y -56.266,Z 90.000,A 0.000,B 0.000,C 180.000,E1 0.000} C_DIS
LIN {X 271.794,Y -42.330,Z 90.000,A 0.000,B 0.000,C 180.000,E1 0.000} C_DIS
LIN {X 273.612,Y -28.283,Z 90.000,A 0.000,B 0.000,C 180.000,E1 0.000} C_DIS
LIN {X 274.705,Y -14.159,Z 90.000,A 0.000,B 0.000,C 180.000,E1 0.000} C_DIS
LIN {X 275.070,Y 0.000,Z 90.000,A 0.000,B 0.000,C 180.000,E1 0.000} C_DIS
LIN {X 274.705,Y 14.159,Z 90.000,A 0.000,B 0.000,C 180.000,E1 0.000} C_DIS
LIN {X 273.612,Y 28.283,Z 90.000,A 0.000,B 0.000,C 180.000,E1 0.000} C_DIS
LIN {X 271.794,Y 42.330,Z 90.000,A 0.000,B 0.000,C 180.000,E1 0.000} C_DIS
LIN {X 269.253,Y 56.266,Z 90.000,A 0.000,B 0.000,C 180.000,E1 0.000} C_DIS
LIN {X 266.000,Y 70.053,Z 90.000,A 0.000,B 0.000,C 180.000,E1 0.000} C_DIS
LIN {X 262.041,Y 83.652,Z 90.000,A 0.000,B 0.000,C 180.000,E1 0.000} C_DIS
LIN {X 257.387,Y 97.031,Z 90.000,A 0.000,B 0.000,C 180.000,E1 0.000} C_DIS
LIN {X 252.050,Y 110.154,Z 90.000,A 0.000,B 0.000,C 180.000,E1 0.000} C_DIS
LIN {X 246.047,Y 122.982,Z 90.000,A 0.000,B 0.000,C 180.000,E1 0.000} C_DIS
LIN {X 239.390,Y 135.485,Z 90.000,A 0.000,B 0.000,C 180.000,E1 0.000} C_DIS
LIN {X 232.097,Y 147.628,Z 90.000,A 0.000,B 0.000,C 180.000,E1 0.000} C_DIS
LIN {X 224.182,Y 159.392,Z 90.000,A 0.000,B 0.000,C 180.000,E1 0.000} C_DIS
LIN {X 215.687,Y 170.711,Z 90.000,A 0.000,B 0.000,C 180.000,E1 0.000} C_DIS
LIN {X 206.614,Y 181.588,Z 90.000,A 0.000,B 0.000,C 180.000,E1 0.000} C_DIS
LIN {X 196.992,Y 191.983,Z 90.000,A 0.000,B 0.000,C 180.000,E1 0.000} C_DIS
LIN {X 186.848,Y 201.870,Z 90.000,A 0.000,B 0.000,C 180.000,E1 0.000} C_DIS
LIN {X 176.208,Y 211.220,Z 90.000,A 0.000,B 0.000,C 180.000,E1 0.000} C_DIS
LIN {X 165.101,Y 220.011,Z 90.000,A 0.000,B 0.000,C 180.000,E1 0.000} C_DIS
LIN {X 153.556,Y 228.219,Z 90.000,A 0.000,B 0.000,C 180.000,E1 0.000} C_DIS
LIN {X 141.604,Y 235.821,Z 90.000,A 0.000,B 0.000,C 180.000,E1 0.000} C_DIS
LIN {X 129.276,Y 242.799,Z 90.000,A 0.000,B 0.000,C 180.000,E1 0.000} C_DIS
LIN {X 116.606,Y 249.131,Z 90.000,A 0.000,B 0.000,C 180.000,E1 0.000} C_DIS
LIN {X 103.624,Y 254.805,Z 90.000,A 0.000,B 0.000,C 180.000,E1 0.000} C_DIS
LIN {X 90.373,Y 259.801,Z 90.000,A 0.000,B 0.000,C 180.000,E1 0.000} C_DIS
LIN {X 76.878,Y 264.108,Z 90.000,A 0.000,B 0.000,C 180.000,E1 0.000} C_DIS
LIN {X 63.179,Y 267.716,Z 90.000,A 0.000,B 0.000,C 180.000,E1 0.000} C_DIS
LIN {X 49.316,Y 270.613,Z 90.000,A 0.000,B 0.000,C 180.000,E1 0.000} C_DIS
LIN {X 35.318,Y 272.792,Z 90.000,A 0.000,B 0.000,C 180.000,E1 0.000} C_DIS
LIN {X 21.229,Y 274.249,Z 90.000,A 0.000,B 0.000,C 180.000,E1 0.000} C_DIS
LIN {X 7.082,Y 274.979,Z 90.000,A 0.000,B 0.000,C 180.000,E1 0.000} C_DIS
LIN {X -7.082,Y 274.979,Z 90.000,A 0.000,B 0.000,C 180.000,E1 0.000} C_DIS
LIN {X -21.229,Y 274.249,Z 90.000,A 0.000,B 0.000,C 180.000,E1 0.000} C_DIS
LIN {X -35.318,Y 272.792,Z 90.000,A 0.000,B 0.000,C 180.000,E1 0.000} C_DIS
LIN {X -49.316,Y 270.613,Z 90.000,A 0.000,B 0.000,C 180.000,E1 0.000} C_DIS
LIN {X -63.179,Y 267.716,Z 90.000,A 0.000,B 0.000,C 180.000,E1 0.000} C_DIS
LIN {X -76.878,Y 264.108,Z 90.000,A 0.000,B 0.000,C 180.000,E1 0.000} C_DIS
LIN {X -90.373,Y 259.801,Z 90.000,A 0.000,B 0.000,C 180.000,E1 0.000} C_DIS
LIN {X -103.626,Y 254.804,Z 90.000,A 0.000,B 0.000,C 180.000,E1 0.000} C_DIS
LIN {X -116.606,Y 249.131,Z 90.000,A 0.000,B 0.000,C 180.000,E1 0.000} C_DIS
LIN {X -129.276,Y 242.799,Z 90.000,A 0.000,B 0.000,C 180.000,E1 0.000} C_DIS
LIN {X -141.604,Y 235.821,Z 90.000,A 0.000,B 0.000,C 180.000,E1 0.000} C_DIS
LIN {X -153.556,Y 228.219,Z 90.000,A 0.000,B 0.000,C 180.000,E1 0.000} C_DIS
LIN {X -165.101,Y 220.011,Z 90.000,A 0.000,B 0.000,C 180.000,E1 0.000} C_DIS
LIN {X -176.208,Y 211.220,Z 90.000,A 0.000,B 0.000,C 180.000,E1 0.000} C_DIS
;rapid-leaky
$VEL.CP=0.3
LIN {X -166.251,Y 199.283,Z 90.000,A 0.000,B 0.000,C 180.000,E1 0.000} C_DIS
;bead-perimeter_inner
$VEL.CP=0.69
LIN {X -176.288,Y 190.462,Z 90.000,A 0.000,B 0.000,C 180.000,E1 0.000} C_DIS
LIN {X -185.868,Y 181.125,Z 90.000,A 0.000,B 0.000,C 180.000,E1 0.000} C_DIS
LIN {X -194.937,Y 171.326,Z 90.000,A 0.000,B 0.000,C 180.000,E1 0.000} C_DIS
LIN {X -203.498,Y 161.064,Z 90.000,A 0.000,B 0.000,C 180.000,E1 0.000} C_DIS
LIN {X -211.519,Y 150.374,Z 90.000,A 0.000,B 0.000,C 180.000,E1 0.000} C_DIS
LIN {X -218.981,Y 139.285,Z 90.000,A 0.000,B 0.000,C 180.000,E1 0.000} C_DIS
LIN {X -225.861,Y 127.828,Z 90.000,A 0.000,B 0.000,C 180.000,E1 0.000} C_DIS
LIN {X -232.142,Y 116.032,Z 90.000,A 0.000,B 0.000,C 180.000,E1 0.000} C_DIS
LIN {X -237.806,Y 103.929,Z 90.000,A 0.000,B 0.000,C 180.000,E1 0.000} C_DIS
LIN {X -242.841,Y 91.547,Z 90.000,A 0.000,B 0.000,C 180.000,E1 0.000} C_DIS
LIN {X -247.233,Y 78.924,Z 90.000,A 0.000,B 0.000,C 180.000,E1 0.000} C_DIS
LIN {X -250.968,Y 66.095,Z 90.000,A 0.000,B 0.000,C 180.000,E1 0.000} C_DIS
LIN {X -254.037,Y 53.086,Z 90.000,A 0.000,B 0.000,C 180.000,E1 0.000} C_DIS
LIN {X -256.434,Y 39.937,Z 90.000,A 0.000,B 0.000,C 180.000,E1 0.000} C_DIS
LIN {X -258.149,Y 26.685,Z 90.000,A 0.000,B 0.000,C 180.000,E1 0.000} C_DIS
LIN {X -259.181,Y 13.359,Z 90.000,A 0.000,B 0.000,C 180.000,E1 0.000} C_DIS
LIN {X -259.525,Y 0.000,Z 90.000,A 0.000,B 0.000,C 180.000,E1 0.000} C_DIS
LIN {X -259.181,Y -13.359,Z 90.000,A 0.000,B 0.000,C 180.000,E1 0.000} C_DIS
LIN {X -258.149,Y -26.685,Z 90.000,A 0.000,B 0.000,C 180.000,E1 0.000} C_DIS
LIN {X -256.434,Y -39.937,Z 90.000,A 0.000,B 0.000,C 180.000,E1 0.000} C_DIS
LIN {X -254.037,Y -53.086,Z 90.000,A 0.000,B 0.000,C 180.000,E1 0.000} C_DIS
LIN {X -250.968,Y -66.095,Z 90.000,A 0.000,B 0.000,C 180.000,E1 0.000} C_DIS
LIN {X -247.233,Y -78.924,Z 90.000,A 0.000,B 0.000,C 180.000,E1 0.000} C_DIS
LIN {X -242.841,Y -91.547,Z 90.000,A 0.000,B 0.000,C 180.000,E1 0.000} C_DIS
LIN {X -237.806,Y -103.929,Z 90.000,A 0.000,B 0.000,C 180.000,E1 0.000} C_DIS
LIN {X -232.142,Y -116.032,Z 90.000,A 0.000,B 0.000,C 180.000,E1 0.000} C_DIS
LIN {X -225.861,Y -127.828,Z 90.000,A 0.000,B 0.000,C 180.000,E1 0.000} C_DIS
LIN {X -218.981,Y -139.285,Z 90.000,A 0.000,B 0.000,C 180.000,E1 0.000} C_DIS
LIN {X -211.512,Y -150.384,Z 90.000,A 0.000,B 0.000,C 180.000,E1 0.000} C_DIS
LIN {X -203.498,Y -161.063,Z 90.000,A 0.000,B 0.000,C 180.000,E1 0.000} C_DIS
LIN {X -194.937,Y -171.326,Z 90.000,A 0.000,B 0.000,C 180.000,E1 0.000} C_DIS
LIN {X -185.859,Y -181.134,Z 90.000,A 0.000,B 0.000,C 180.000,E1 0.000} C_DIS
LIN {X -176.288,Y -190.462,Z 90.000,A 0.000,B 0.000,C 180.000,E1 0.000} C_DIS
LIN {X -166.251,Y -199.283,Z 90.000,A 0.000,B 0.000,C 180.000,E1 0.000} C_DIS
LIN {X -155.770,Y -207.577,Z 90.000,A 0.000,B 0.000,C 180.000,E1 0.000} C_DIS
LIN {X -144.878,Y -215.321,Z 90.000,A 0.000,B 0.000,C 180.000,E1 0.000} C_DIS
LIN {X -133.601,Y -222.494,Z 90.000,A 0.000,B 0.000,C 180.000,E1 0.000} C_DIS
LIN {X -121.970,Y -229.078,Z 90.000,A 0.000,B 0.000,C 180.000,E1 0.000} C_DIS
LIN {X -110.016,Y -235.052,Z 90.000,A 0.000,B 0.000,C 180.000,E1 0.000} C_DIS
LIN {X -97.768,Y -240.405,Z 90.000,A 0.000,B 0.000,C 180.000,E1 0.000} C_DIS
LIN {X -85.267,Y -245.118,Z 90.000,A 0.000,B 0.000,C 180.000,E1 0.000} C_DIS
LIN {X -72.533,Y -249.182,Z 90.000,A 0.000,B 0.000,C 180.000,E1 0.000} C_DIS
LIN {X -59.608,Y -252.587,Z 90.000,A 0.000,B 0.000,C 180.000,E1 0.000} C_DIS
LIN {X -46.529,Y -255.320,Z 90.000,A 0.000,B 0.000,C 180.000,E1 0.000} C_DIS
LIN {X -33.322,Y -257.376,Z 90.000,A 0.000,B 0.000,C 180.000,E1 0.000} C_DIS
LIN {X -20.028,Y -258.751,Z 90.000,A 0.000,B 0.000,C 180.000,E1 0.000} C_DIS
LIN {X -6.682,Y -259.439,Z 90.000,A 0.000,B 0.000,C 180.000,E1 0.000} C_DIS
LIN {X 6.682,Y -259.439,Z 90.000,A 0.000,B 0.000,C 180.000,E1 0.000} C_DIS
LIN {X 20.028,Y -258.751,Z 90.000,A 0.000,B 0.000,C 180.000,E1 0.000} C_DIS
LIN {X 33.322,Y -257.376,Z 90.000,A 0.000,B 0.000,C 180.000,E1 0.000} C_DIS
LIN {X 46.529,Y -255.320,Z 90.000,A 0.000,B 0.000,C 180.000,E1 0.000} C_DIS
LIN {X 59.608,Y -252.587,Z 90.000,A 0.000,B 0.000,C 180.000,E1 0.000} C_DIS
LIN {X 72.533,Y -249.182,Z 90.000,A 0.000,B 0.000,C 180.000,E1 0.000} C_DIS
LIN {X 85.267,Y -245.118,Z 90.000,A 0.000,B 0.000,C 180.000,E1 0.000} C_DIS
LIN {X 97.769,Y -240.405,Z 90.000,A 0.000,B 0.000,C 180.000,E1 0.000} C_DIS
LIN {X 110.016,Y -235.052,Z 90.000,A 0.000,B 0.000,C 180.000,E1 0.000} C_DIS
LIN {X 121.970,Y -229.078,Z 90.000,A 0.000,B 0.000,C 180.000,E1 0.000} C_DIS
LIN {X 133.601,Y -222.494,Z 90.000,A 0.000,B 0.000,C 180.000,E1 0.000} C_DIS
LIN {X 144.878,Y -215.321,Z 90.000,A 0.000,B 0.000,C 180.000,E1 0.000} C_DIS
LIN {X 155.770,Y -207.577,Z 90.000,A 0.000,B 0.000,C 180.000,E1 0.000} C_DIS
LIN {X 166.251,Y -199.283,Z 90.000,A 0.000,B 0.000,C 180.000,E1 0.000} C_DIS
LIN {X 176.288,Y -190.462,Z 90.000,A 0.000,B 0.000,C 180.000,E1 0.000} C_DIS
LIN {X 185.868,Y -181.125,Z 90.000,A 0.000,B 0.000,C 180.000,E1 0.000} C_DIS
LIN {X 194.937,Y -171.326,Z 90.000,A 0.000,B 0.000,C 180.000,E1 0.000} C_DIS
LIN {X 203.498,Y -161.064,Z 90.000,A 0.000,B 0.000,C 180.000,E1 0.000} C_DIS
LIN {X 211.519,Y -150.374,Z 90.000,A 0.000,B 0.000,C 180.000,E1 0.000} C_DIS
LIN {X 218.981,Y -139.285,Z 90.000,A 0.000,B 0.000,C 180.000,E1 0.000} C_DIS
LIN {X 225.861,Y -127.828,Z 90.000,A 0.000,B 0.000,C 180.000,E1 0.000} C_DIS
LIN {X 232.142,Y -116.032,Z 90.000,A 0.000,B 0.000,C 180.000,E1 0.000} C_DIS
LIN {X 237.806,Y -103.929,Z 90.000,A 0.000,B 0.000,C 180.000,E1 0.000} C_DIS
LIN {X 242.841,Y -91.547,Z 90.000,A 0.000,B 0.000,C 180.000,E1 0.000} C_DIS
LIN {X 247.233,Y -78.924,Z 90.000,A 0.000,B 0.000,C 180.000,E1 0.000} C_DIS
LIN {X 250.968,Y -66.095,Z 90.000,A 0.000,B 0.000,C 180.000,E1 0.000} C_DIS
LIN {X 254.037,Y -53.086,Z 90.000,A 0.000,B 0.000,C 180.000,E1 0.000} C_DIS
LIN {X 256.434,Y -39.937,Z 90.000,A 0.000,B 0.000,C 180.000,E1 0.000} C_DIS
LIN {X 258.149,Y -26.685,Z 90.000,A 0.000,B 0.000,C 180.000,E1 0.000} C_DIS
LIN {X 259.181,Y -13.359,Z 90.000,A 0.000,B 0.000,C 180.000,E1 0.000} C_DIS
LIN {X 259.525,Y 0.000,Z 90.000,A 0.000,B 0.000,C 180.000,E1 0.000} C_DIS
LIN {X 259.181,Y 13.359,Z 90.000,A 0.000,B 0.000,C 180.000,E1 0.000} C_DIS
LIN {X 258.149,Y 26.685,Z 90.000,A 0.000,B 0.000,C 180.000,E1 0.000} C_DIS
LIN {X 256.434,Y 39.937,Z 90.000,A 0.000,B 0.000,C 180.000,E1 0.000} C_DIS
LIN {X 254.037,Y 53.086,Z 90.000,A 0.000,B 0.000,C 180.000,E1 0.000} C_DIS
LIN {X 250.968,Y 66.095,Z 90.000,A 0.000,B 0.000,C 180.000,E1 0.000} C_DIS
LIN {X 247.233,Y 78.924,Z 90.000,A 0.000,B 0.000,C 180.000,E1 0.000} C_DIS
LIN {X 242.841,Y 91.547,Z 90.000,A 0.000,B 0.000,C 180.000,E1 0.000} C_DIS
LIN {X 237.806,Y 103.929,Z 90.000,A 0.000,B 0.000,C 180.000,E1 0.000} C_DIS
LIN {X 232.142,Y 116.032,Z 90.000,A 0.000,B 0.000,C 180.000,E1 0.000} C_DIS
LIN {X 225.861,Y 127.828,Z 90.000,A 0.000,B 0.000,C 180.000,E1 0.000} C_DIS
LIN {X 218.981,Y 139.285,Z 90.000,A 0.000,B 0.000,C 180.000,E1 0.000} C_DIS
LIN {X 211.512,Y 150.384,Z 90.000,A 0.000,B 0.000,C 180.000,E1 0.000} C_DIS
LIN {X 203.498,Y 161.063,Z 90.000,A 0.000,B 0.000,C 180.000,E1 0.000} C_DIS
LIN {X 194.937,Y 171.326,Z 90.000,A 0.000,B 0.000,C 180.000,E1 0.000} C_DIS
LIN {X 185.859,Y 181.134,Z 90.000,A 0.000,B 0.000,C 180.000,E1 0.000} C_DIS
LIN {X 176.288,Y 190.462,Z 90.000,A 0.000,B 0.000,C 180.000,E1 0.000} C_DIS
LIN {X 166.251,Y 199.283,Z 90.000,A 0.000,B 0.000,C 180.000,E1 0.000} C_DIS
LIN {X 155.770,Y 207.577,Z 90.000,A 0.000,B 0.000,C 180.000,E1 0.000} C_DIS
LIN {X 144.878,Y 215.321,Z 90.000,A 0.000,B 0.000,C 180.000,E1 0.000} C_DIS
LIN {X 133.601,Y 222.494,Z 90.000,A 0.000,B 0.000,C 180.000,E1 0.000} C_DIS
LIN {X 121.970,Y 229.078,Z 90.000,A 0.000,B 0.000,C 180.000,E1 0.000} C_DIS
LIN {X 110.016,Y 235.052,Z 90.000,A 0.000,B 0.000,C 180.000,E1 0.000} C_DIS
LIN {X 97.768,Y 240.405,Z 90.000,A 0.000,B 0.000,C 180.000,E1 0.000} C_DIS
LIN {X 85.267,Y 245.118,Z 90.000,A 0.000,B 0.000,C 180.000,E1 0.000} C_DIS
LIN {X 72.533,Y 249.182,Z 90.000,A 0.000,B 0.000,C 180.000,E1 0.000} C_DIS
LIN {X 59.608,Y 252.587,Z 90.000,A 0.000,B 0.000,C 180.000,E1 0.000} C_DIS
LIN {X 46.529,Y 255.320,Z 90.000,A 0.000,B 0.000,C 180.000,E1 0.000} C_DIS
LIN {X 33.322,Y 257.376,Z 90.000,A 0.000,B 0.000,C 180.000,E1 0.000} C_DIS
LIN {X 20.028,Y 258.751,Z 90.000,A 0.000,B 0.000,C 180.000,E1 0.000} C_DIS
LIN {X 6.682,Y 259.439,Z 90.000,A 0.000,B 0.000,C 180.000,E1 0.000} C_DIS
LIN {X -6.682,Y 259.439,Z 90.000,A 0.000,B 0.000,C 180.000,E1 0.000} C_DIS
LIN {X -20.028,Y 258.751,Z 90.000,A 0.000,B 0.000,C 180.000,E1 0.000} C_DIS
LIN {X -33.322,Y 257.376,Z 90.000,A 0.000,B 0.000,C 180.000,E1 0.000} C_DIS
LIN {X -46.529,Y 255.320,Z 90.000,A 0.000,B 0.000,C 180.000,E1 0.000} C_DIS
LIN {X -59.608,Y 252.587,Z 90.000,A 0.000,B 0.000,C 180.000,E1 0.000} C_DIS
LIN {X -72.533,Y 249.182,Z 90.000,A 0.000,B 0.000,C 180.000,E1 0.000} C_DIS
LIN {X -85.267,Y 245.118,Z 90.000,A 0.000,B 0.000,C 180.000,E1 0.000} C_DIS
LIN {X -97.769,Y 240.405,Z 90.000,A 0.000,B 0.000,C 180.000,E1 0.000} C_DIS
LIN {X -110.016,Y 235.052,Z 90.000,A 0.000,B 0.000,C 180.000,E1 0.000} C_DIS
LIN {X -121.970,Y 229.078,Z 90.000,A 0.000,B 0.000,C 180.000,E1 0.000} C_DIS
LIN {X -133.601,Y 222.494,Z 90.000,A 0.000,B 0.000,C 180.000,E1 0.000} C_DIS
LIN {X -144.878,Y 215.321,Z 90.000,A 0.000,B 0.000,C 180.000,E1 0.000} C_DIS
LIN {X -155.770,Y 207.577,Z 90.000,A 0.000,B 0.000,C 180.000,E1 0.000} C_DIS
LIN {X -166.251,Y 199.283,Z 90.000,A 0.000,B 0.000,C 180.000,E1 0.000} C_DIS
;rapid-leaky
$VEL.CP=0.3
LIN {X 237.442,Y 45.088,Z 90.000,A 0.000,B 0.000,C 180.000,E1 0.000} C_DIS
;bead-sparse_infill
$VEL.CP=0.69
LIN {X 45.043,Y 237.487,Z 90.000,A 0.000,B 0.000,C 180.000,E1 0.000} C_DIS
LIN {X 43.345,Y 237.842,Z 90.000,A 0.000,B 0.000,C 180.000,E1 0.000} C_DIS
LIN {X 31.041,Y 239.757,Z 90.000,A 0.000,B 0.000,C 180.000,E1 0.000} C_DIS
LIN {X 18.657,Y 241.038,Z 90.000,A 0.000,B 0.000,C 180.000,E1 0.000} C_DIS
LIN {X 6.224,Y 241.679,Z 90.000,A 0.000,B 0.000,C 180.000,E1 0.000} C_DIS
LIN {X -6.224,Y 241.679,Z 90.000,A 0.000,B 0.000,C 180.000,E1 0.000} C_DIS
LIN {X -18.657,Y 241.038,Z 90.000,A 0.000,B 0.000,C 180.000,E1 0.000} C_DIS
LIN {X -31.041,Y 239.757,Z 90.000,A 0.000,B 0.000,C 180.000,E1 0.000} C_DIS
LIN {X -43.345,Y 237.842,Z 90.000,A 0.000,B 0.000,C 180.000,E1 0.000} C_DIS
LIN {X -55.527,Y 235.296,Z 90.000,A 0.000,B 0.000,C 180.000,E1 0.000} C_DIS
LIN {X -67.568,Y 232.124,Z 90.000,A 0.000,B 0.000,C 180.000,E1 0.000} C_DIS
LIN {X -79.430,Y 228.338,Z 90.000,A 0.000,B 0.000,C 180.000,E1 0.000} C_DIS
LIN {X -91.076,Y 223.948,Z 90.000,A 0.000,B 0.000,C 180.000,E1 0.000} C_DIS
LIN {X -96.170,Y 221.722,Z 90.000,A 0.000,B 0.000,C 180.000,E1 0.000} C_DIS
LIN {X 221.770,Y -96.218,Z 90.000,A 0.000,B 0.000,C 180.000,E1 0.000} C_DIS
LIN {X 221.527,Y -96.815,Z 90.000,A 0.000,B 0.000,C 180.000,E1 0.000} C_DIS
LIN {X 216.250,Y -108.089,Z 90.000,A 0.000,B 0.000,C 180.000,E1 0.000} C_DIS
LIN {X 210.400,Y -119.077,Z 90.000,A 0.000,B 0.000,C 180.000,E1 0.000} C_DIS
LIN {X 203.991,Y -129.750,Z 90.000,A 0.000,B 0.000,C 180.000,E1 0.000} C_DIS
LIN {X 197.040,Y -140.080,Z 90.000,A 0.000,B 0.000,C 180.000,E1 0.000} C_DIS
LIN {X 189.567,Y -150.038,Z 90.000,A 0.000,B 0.000,C 180.000,E1 0.000} C_DIS
LIN {X 181.592,Y -159.599,Z 90.000,A 0.000,B 0.000,C 180.000,E1 0.000} C_DIS
LIN {X 173.145,Y -168.726,Z 90.000,A 0.000,B 0.000,C 180.000,E1 0.000} C_DIS
LIN {X 164.220,Y -177.424,Z 90.000,A 0.000,B 0.000,C 180.000,E1 0.000} C_DIS
LIN {X 154.871,Y -185.641,Z 90.000,A 0.000,B 0.000,C 180.000,E1 0.000} C_DIS
LIN {X 154.505,Y -185.930,Z 90.000,A 0.000,B 0.000,C 180.000,E1 0.000} C_DIS
LIN {X -185.882,Y 154.456,Z 90.000,A 0.000,B 0.000,C 180.000,E1 0.000} C_DIS
LIN {X -189.567,Y 150.038,Z 90.000,A 0.000,B 0.000,C 180.000,E1 0.000} C_DIS
LIN {X -197.040,Y 140.080,Z 90.000,A 0.000,B 0.000,C 180.000,E1 0.000} C_DIS
LIN {X -203.991,Y 129.750,Z 90.000,A 0.000,B 0.000,C 180.000,E1 0.000} C_DIS
LIN {X -210.400,Y 119.077,Z 90.000,A 0.000,B 0.000,C 180.000,E1 0.000} C_DIS
LIN {X -216.250,Y 108.089,Z 90.000,A 0.000,B 0.000,C 180.000,E1 0.000} C_DIS
LIN {X -221.527,Y 96.815,Z 90.000,A 0.000,B 0.000,C 180.000,E1 0.000} C_DIS
LIN {X -226.217,Y 85.281,Z 90.000,A 0.000,B 0.000,C 180.000,E1 0.000} C_DIS
LIN {X -230.308,Y 73.520,Z 90.000,A 0.000,B 0.000,C 180.000,E1 0.000} C_DIS
LIN {X -233.787,Y 61.571,Z 90.000,A 0.000,B 0.000,C 180.000,E1 0.000} C_DIS
LIN {X -236.646,Y 49.452,Z 90.000,A 0.000,B 0.000,C 180.000,E1 0.000} C_DIS
LIN {X -236.833,Y 48.429,Z 90.000,A 0.000,B 0.000,C 180.000,E1 0.000} C_DIS
LIN {X 48.385,Y -236.788,Z 90.000,A 0.000,B 0.000,C 180.000,E1 0.000} C_DIS
;rapid-leaky
$VEL.CP=0.3
LIN {X 151.650,Y 225.387,Z 100.000,A 0.000,B 0.000,C 180.000,E1 0.000} C_DIS
;bead-perimeter_outer
$VEL.CP=0.68
LIN {X 139.846,Y 232.895,Z 100.000,A 0.000,B 0.000,C 180.000,E1 0.000} C_DIS
LIN {X 127.671,Y 239.785,Z 100.000,A 0.000,B 0.000,C 180.000,E1 0.000} C_DIS
LIN {X 115.159,Y 246.039,Z 100.000,A 0.000,B 0.000,C 180.000,E1 0.000} C_DIS
LIN {X 102.340,Y 251.641,Z 100.000,A 0.000,B 0.000,C 180.000,E1 0.000} C_DIS
LIN {X 89.250,Y 256.576,Z 100.000,A 0.000,B 0.000,C 180.000,E1 0.000} C_DIS
LIN {X 75.923,Y 260.831,Z 100.000,A 0.000,B 0.000,C 180.000,E1 0.000} C_DIS
LIN {X 62.396,Y 264.393,Z 100.000,A 0.000,B 0.000,C 180.000,E1 0.000} C_DIS
LIN {X 48.702,Y 267.254,Z 100.000,A 0.000,B 0.000,C 180.000,E1 0.000} C_DIS
LIN {X 34.880,Y 269.407,Z 100.000,A 0.000,B 0.000,C 180.000,E1 0.000} C_DIS
LIN {X 20.965,Y 270.845,Z 100.000,A 0.000,B 0.000,C 180.000,E1 0.000} C_DIS
LIN {X 6.995,Y 271.566,Z 100.000,A 0.000,B 0.000,C 180.000,E1 0.000} C_DIS
LIN {X -6.995,Y 271.566,Z 100.000,A 0.000,B 0.000,C 180.000,E1 0.000} C_DIS
LIN {X -16.957,Y 271.053,Z 100.000,A 0.000,B 0.000,C 180.000,E1 0.000} C_DIS
LIN {X -20.964,Y 270.846,Z 100.000,A 0.000,B 0.000,C 180.000,E1 0.000} C_DIS
LIN {X -34.880,Y 269.407,Z 100.000,A 0.000,B 0.000,C 180.000,E1 0.000} C_DIS
LIN {X -48.702,Y 267.254,Z 100.000,A 0.000,B 0.000,C 180.000,E1 0.000} C_DIS
LIN {X -62.396,Y 264.393,Z 100.000,A 0.000,B 0.000,C 180.000,E1 0.000} C_DIS
LIN {X -75.923,Y 260.831,Z 100.000,A 0.000,B 0.000,C 180.000,E1 0.000} C_DIS
LIN {X -89.250,Y 256.576,Z 100.000,A 0.000,B 0.000,C 180.000,E1 0.000} C_DIS
LIN {X -102.340,Y 251.641,Z 100.000,A 0.000,B 0.000,C 180.000,E1 0.000} C_DIS
LIN {X -115.159,Y 246.039,Z 100.000,A 0.000,B 0.000,C 180.000,E1 0.000} C_DIS
LIN {X -127.671,Y 239.785,Z 100.000,A 0.000,B 0.000,C 180.000,E1 0.000} C_DIS
LIN {X -139.846,Y 232.895,Z 100.000,A 0.000,B 0.000,C 180.000,E1 0.000} C_DIS
LIN {X -151.650,Y 225.387,Z 100.000,A 0.000,B 0.000,C 180.000,E1 0.000} C_DIS
LIN {X -163.051,Y 217.281,Z 100.000,A 0.000,B 0.000,C 180.000,E1 0.000} C_DIS
LIN {X -174.021,Y 208.599,Z 100.000,A 0.000,B 0.000,C 180.000,E1 0.000} C_DIS
LIN {X -184.529,Y 199.364,Z 100.000,A 0.000,B 0.000,C 180.000,E1 0.000} C_DIS
LIN {X -194.547,Y 189.601,Z 100.000,A 0.000,B 0.000,C 180.000,E1 0.000} C_DIS
LIN {X -204.049,Y 179.334,Z 100.000,A 0.000,B 0.000,C 180.000,E1 0.000} C_DIS
LIN {X -213.010,Y 168.592,Z 100.000,A 0.000,B 0.000,C 180.000,E1 0.000} C_DIS
LIN {X -221.407,Y 157.403,Z 100.000,A 0.000,B 0.000,C 180.000,E1 0.000} C_DIS
LIN {X -229.217,Y 145.797,Z 100.000,A 0.000,B 0.000,C 180.000,E1 0.000} C_DIS
LIN {X -236.418,Y 133.803,Z 100.000,A 0.000,B 0.000,C 180.000,E1 0.000} C_DIS
LIN {X -242.993,Y 121.456,Z 100.000,A 0.000,B 0.000,C 180.000,E1 0.000} C_DIS
LIN {X -248.923,Y 108.786,Z 100.000,A 0.000,B 0.000,C 180.000,E1 0.000} C_DIS
LIN {X -254.193,Y 95.827,Z 100.000,A 0.000,B 0.000,C 180.000,E1 0.000} C_DIS
LIN {X -258.789,Y 82.614,Z 100.000,A 0.000,B 0.000,C 180.000,E1 0.000} C_DIS
LIN {X -262.699,Y 69.184,Z 100.000,A 0.000,B 0.000,C 180.000,E1 0.000} C_DIS
LIN {X -265.911,Y 55.568,Z 100.000,A 0.000,B 0.000,C 180.000,E1 0.000} C_DIS
LIN {X -268.420,Y 41.805,Z 100.000,A 0.000,B 0.000,C 180.000,E1 0.000} C_DIS
LIN {X -270.216,Y 27.932,Z 100.000,A 0.000,B 0.000,C 180.000,E1 0.000} C_DIS
LIN {X -271.296,Y 13.984,Z 100.000,A 0.000,B 0.000,C 180.000,E1 0.000} C_DIS
LIN {X -271.656,Y 0.000,Z 100.000,A 0.000,B 0.000,C 180.000,E1 0.000} C_DIS
LIN {X -271.296,Y -13.984,Z 100.000,A 0.000,B 0.000,C 180.000,E1 0.000} C_DIS
LIN {X -270.216,Y -27.932,Z 100.000,A 0.000,B 0.000,C 180.000,E1 0.000} C_DIS
LIN {X -268.420,Y -41.805,Z 100.000,A 0.000,B 0.000,C 180.000,E1 0.000} C_DIS
LIN {X -265.911,Y -55.568,Z 100.000,A 0.000,B 0.000,C 180.000,E1 0.000} C_DIS
LIN {X -262.699,Y -69.184,Z 100.000,A 0.000,B 0.000,C 180.000,E1 0.000} C_DIS
LIN {X -258.789,Y -82.614,Z 100.000,A 0.000,B 0.000,C 180.000,E1 0.000} C_DIS
LIN {X -254.193,Y -95.827,Z 100.000,A 0.000,B 0.000,C 180.000,E1 0.000} C_DIS
LIN {X -248.923,Y -108.786,Z 100.000,A 0.000,B 0.000,C 180.000,E1 0.000} C_DIS
LIN {X -242.993,Y -121.456,Z 100.000,A 0.000,B 0.000,C 180.000,E1 0.000} C_DIS
LIN {X -236.419,Y -133.803,Z 100.000,A 0.000,B 0.000,C 180.000,E1 0.000} C_DIS
LIN {X -229.217,Y -145.797,Z 100.000,A 0.000,B 0.000,C 180.000,E1 0.000} C_DIS
LIN {X -221.407,Y -157.403,Z 100.000,A 0.000,B 0.000,C 180.000,E1 0.000} C_DIS
LIN {X -213.010,Y -168.592,Z 100.000,A 0.000,B 0.000,C 180.000,E1 0.000} C_DIS
LIN {X -204.049,Y -179.334,Z 100.000,A 0.000,B 0.000,C 180.000,E1 0.000} C_DIS
LIN {X -194.547,Y -189.601,Z 100.000,A 0.000,B 0.000,C 180.000,E1 0.000} C_DIS
LIN {X -184.529,Y -199.364,Z 100.000,A 0.000,B 0.000,C 180.000,E1 0.000} C_DIS
LIN {X -174.021,Y -208.599,Z 100.000,A 0.000,B 0.000,C 180.000,E1 0.000} C_DIS
LIN {X -163.051,Y -217.281,Z 100.000,A 0.000,B 0.000,C 180.000,E1 0.000} C_DIS
LIN {X -151.650,Y -225.387,Z 100.000,A 0.000,B 0.000,C 180.000,E1 0.000} C_DIS
LIN {X -139.846,Y -232.895,Z 100.000,A 0.000,B 0.000,C 180.000,E1 0.000} C_DIS
LIN {X -127.671,Y -239.785,Z 100.000,A 0.000,B 0.000,C 180.000,E1 0.000} C_DIS
LIN {X -115.159,Y -246.039,Z 100.000,A 0.000,B 0.000,C 180.000,E1 0.000} C_DIS
LIN {X -102.340,Y -251.641,Z 100.000,A 0.000,B 0.000,C 180.000,E1 0.000} C_DIS
LIN {X -89.250,Y -256.576,Z 100.000,A 0.000,B 0.000,C 180.000,E1 0.000} C_DIS
LIN {X -75.923,Y -260.831,Z 100.000,A 0.000,B 0.000,C 180.000,E1 0.000} C_DIS
LIN {X -62.396,Y -264.393,Z 100.000,A 0.000,B 0.000,C 180.000,E1 0.000} C_DIS
LIN {X -48.702,Y -267.254,Z 100.000,A 0.000,B 0.000,C 180.000,E1 0.000} C_DIS
LIN {X -34.880,Y -269.407,Z 100.000,A 0.000,B 0.000,C 180.000,E1 0.000} C_DIS
LIN {X -20.965,Y -270.845,Z 100.000,A 0.000,B 0.000,C 180.000,E1 0.000} C_DIS
LIN {X -6.995,Y -271.566,Z 100.000,A 0.000,B 0.000,C 180.000,E1 0.000} C_DIS
LIN {X 6.995,Y -271.566,Z 100.000,A 0.000,B 0.000,C 180.000,E1 0.000} C_DIS
LIN {X 16.957,Y -271.053,Z 100.000,A 0.000,B 0.000,C 180.000,E1 0.000} C_DIS
LIN {X 20.964,Y -270.846,Z 100.000,A 0.000,B 0.000,C 180.000,E1 0.000} C_DIS
LIN {X 34.880,Y -269.407,Z 100.000,A 0.000,B 0.000,C 180.000,E1 0.000} C_DIS
LIN {X 48.702,Y -267.254,Z 100.000,A 0.000,B 0.000,C 180.000,E1 0.000} C_DIS
LIN {X 62.396,Y -264.393,Z 100.000,A 0.000,B 0.000,C 180.000,E1 0.000} C_DIS
LIN {X 75.923,Y -260.831,Z 100.000,A 0.000,B 0.000,C 180.000,E1 0.000} C_DIS
LIN {X 89.250,Y -256.576,Z 100.000,A 0.000,B 0.000,C 180.000,E1 0.000} C_DIS
LIN {X 102.340,Y -251.641,Z 100.000,A 0.000,B 0.000,C 180.000,E1 0.000} C_DIS
LIN {X 115.159,Y -246.039,Z 100.000,A 0.000,B 0.000,C 180.000,E1 0.000} C_DIS
LIN {X 127.671,Y -239.785,Z 100.000,A 0.000,B 0.000,C 180.000,E1 0.000} C_DIS
LIN {X 139.846,Y -232.895,Z 100.000,A 0.000,B 0.000,C 180.000,E1 0.000} C_DIS
LIN {X 151.650,Y -225.387,Z 100.000,A 0.000,B 0.000,C 180.000,E1 0.000} C_DIS
LIN {X 163.051,Y -217.281,Z 100.000,A 0.000,B 0.000,C 180.000,E1 0.000} C_DIS
LIN {X 174.021,Y -208.599,Z 100.000,A 0.000,B 0.000,C 180.000,E1 0.000} C_DIS
LIN {X 184.529,Y -199.364,Z 100.000,A 0.000,B 0.000,C 180.000,E1 0.000} C_DIS
LIN {X 194.547,Y -189.601,Z 100.000,A 0.000,B 0.000,C 180.000,E1 0.000} C_DIS
LIN {X 204.049,Y -179.334,Z 100.000,A 0.000,B 0.000,C 180.000,E1 0.000} C_DIS
LIN {X 213.010,Y -168.592,Z 100.000,A 0.000,B 0.000,C 180.000,E1 0.000} C_DIS
LIN {X 221.407,Y -157.403,Z 100.000,A 0.000,B 0.000,C 180.000,E1 0.000} C_DIS
LIN {X 229.217,Y -145.797,Z 100.000,A 0.000,B 0.000,C 180.000,E1 0.000} C_DIS
LIN {X 236.418,Y -133.803,Z 100.000,A 0.000,B 0.000,C 180.000,E1 0.000} C_DIS
LIN {X 242.993,Y -121.456,Z 100.000,A 0.000,B 0.000,C 180.000,E1 0.000} C_DIS
LIN {X 248.923,Y -108.786,Z 100.000,A 0.000,B 0.000,C 180.000,E1 0.000} C_DIS
LIN {X 254.193,Y -95.827,Z 100.000,A 0.000,B 0.000,C 180.000,E1 0.000} C_DIS
LIN {X 258.789,Y -82.614,Z 100.000,A 0.000,B 0.000,C 180.000,E1 0.000} C_DIS
LIN {X 262.699,Y -69.184,Z 100.000,A 0.000,B 0.000,C 180.000,E1 0.000} C_DIS
LIN {X 265.911,Y -55.568,Z 100.000,A 0.000,B 0.000,C 180.000,E1 0.000} C_DIS
LIN {X 268.420,Y -41.805,Z 100.000,A 0.000,B 0.000,C 180.000,E1 0.000} C_DIS
LIN {X 270.216,Y -27.932,Z 100.000,A 0.000,B 0.000,C 180.000,E1 0.000} C_DIS
LIN {X 271.296,Y -13.984,Z 100.000,A 0.000,B 0.000,C 180.000,E1 0.000} C_DIS
LIN {X 271.656,Y 0.000,Z 100.000,A 0.000,B 0.000,C 180.000,E1 0.000} C_DIS
LIN {X 271.296,Y 13.984,Z 100.000,A 0.000,B 0.000,C 180.000,E1 0.000} C_DIS
LIN {X 270.216,Y 27.932,Z 100.000,A 0.000,B 0.000,C 180.000,E1 0.000} C_DIS
LIN {X 268.420,Y 41.805,Z 100.000,A 0.000,B 0.000,C 180.000,E1 0.000} C_DIS
LIN {X 265.911,Y 55.568,Z 100.000,A 0.000,B 0.000,C 180.000,E1 0.000} C_DIS
LIN {X 262.699,Y 69.184,Z 100.000,A 0.000,B 0.000,C 180.000,E1 0.000} C_DIS
LIN {X 258.789,Y 82.614,Z 100.000,A 0.000,B 0.000,C 180.000,E1 0.000} C_DIS
LIN {X 254.193,Y 95.827,Z 100.000,A 0.000,B 0.000,C 180.000,E1 0.000} C_DIS
LIN {X 248.923,Y 108.786,Z 100.000,A 0.000,B 0.000,C 180.000,E1 0.000} C_DIS
LIN {X 242.993,Y 121.456,Z 100.000,A 0.000,B 0.000,C 180.000,E1 0.000} C_DIS
LIN {X 236.419,Y 133.803,Z 100.000,A 0.000,B 0.000,C 180.000,E1 0.000} C_DIS
LIN {X 229.217,Y 145.797,Z 100.000,A 0.000,B 0.000,C 180.000,E1 0.000} C_DIS
LIN {X 221.407,Y 157.403,Z 100.000,A 0.000,B 0.000,C 180.000,E1 0.000} C_DIS
LIN {X 213.010,Y 168.592,Z 100.000,A 0.000,B 0.000,C 180.000,E1 0.000} C_DIS
LIN {X 204.049,Y 179.334,Z 100.000,A 0.000,B 0.000,C 180.000,E1 0.000} C_DIS
LIN {X 194.547,Y 189.601,Z 100.000,A 0.000,B 0.000,C 180.000,E1 0.000} C_DIS
LIN {X 184.529,Y 199.364,Z 100.000,A 0.000,B 0.000,C 180.000,E1 0.000} C_DIS
LIN {X 174.021,Y 208.599,Z 100.000,A 0.000,B 0.000,C 180.000,E1 0.000} C_DIS
LIN {X 163.051,Y 217.281,Z 100.000,A 0.000,B 0.000,C 180.000,E1 0.000} C_DIS
LIN {X 151.650,Y 225.387,Z 100.000,A 0.000,B 0.000,C 180.000,E1 0.000} C_DIS
;rapid-leaky
$VEL.CP=0.3
LIN {X 142.972,Y 212.489,Z 100.000,A 0.000,B 0.000,C 180.000,E1 0.000} C_DIS
;bead-perimeter_inner
$VEL.CP=0.68
LIN {X 131.844,Y 219.568,Z 100.000,A 0.000,B 0.000,C 180.000,E1 0.000} C_DIS
LIN {X 120.365,Y 226.064,Z 100.000,A 0.000,B 0.000,C 180.000,E1 0.000} C_DIS
LIN {X 108.569,Y 231.960,Z 100.000,A 0.000,B 0.000,C 180.000,E1 0.000} C_DIS
LIN {X 96.484,Y 237.241,Z 100.000,A 0.000,B 0.000,C 180.000,E1 0.000} C_DIS
LIN {X 84.142,Y 241.894,Z 100.000,A 0.000,B 0.000,C 180.000,E1 0.000} C_DIS
LIN {X 71.579,Y 245.905,Z 100.000,A 0.000,B 0.000,C 180.000,E1 0.000} C_DIS
LIN {X 58.826,Y 249.263,Z 100.000,A 0.000,B 0.000,C 180.000,E1 0.000} C_DIS
LIN {X 45.916,Y 251.961,Z 100.000,A 0.000,B 0.000,C 180.000,E1 0.000} C_DIS
LIN {X 32.884,Y 253.991,Z 100.000,A 0.000,B 0.000,C 180.000,E1 0.000} C_DIS
LIN {X 19.765,Y 255.347,Z 100.000,A 0.000,B 0.000,C 180.000,E1 0.000} C_DIS
LIN {X 6.594,Y 256.026,Z 100.000,A 0.000,B 0.000,C 180.000,E1 0.000} C_DIS
LIN {X -6.595,Y 256.026,Z 100.000,A 0.000,B 0.000,C 180.000,E1 0.000} C_DIS
LIN {X -16.157,Y 255.533,Z 100.000,A 0.000,B 0.000,C 180.000,E1 0.000} C_DIS
LIN {X -19.764,Y 255.347,Z 100.000,A 0.000,B 0.000,C 180.000,E1 0.000} C_DIS
LIN {X -32.884,Y 253.991,Z 100.000,A 0.000,B 0.000,C 180.000,E1 0.000} C_DIS
LIN {X -45.916,Y 251.961,Z 100.000,A 0.000,B 0.000,C 180.000,E1 0.000} C_DIS
LIN {X -58.826,Y 249.263,Z 100.000,A 0.000,B 0.000,C 180.000,E1 0.000} C_DIS
LIN {X -71.579,Y 245.905,Z 100.000,A 0.000,B 0.000,C 180.000,E1 0.000} C_DIS
LIN {X -84.142,Y 241.894,Z 100.000,A 0.000,B 0.000,C 180.000,E1 0.000} C_DIS
LIN {X -96.484,Y 237.241,Z 100.000,A 0.000,B 0.000,C 180.000,E1 0.000} C_DIS
LIN {X -108.569,Y 231.960,Z 100.000,A 0.000,B 0.000,C 180.000,E1 0.000} C_DIS
LIN {X -120.365,Y 226.064,Z 100.000,A 0.000,B 0.000,C 180.000,E1 0.000} C_DIS
LIN {X -131.844,Y 219.568,Z 100.000,A 0.000,B 0.000,C 180.000,E1 0.000} C_DIS
LIN {X -142.972,Y 212.489,Z 100.000,A 0.000,B 0.000,C 180.000,E1 0.000} C_DIS
LIN {X -153.721,Y 204.847,Z 100.000,A 0.000,B 0.000,C 180.000,E1 0.000} C_DIS
LIN {X -164.063,Y 196.662,Z 100.000,A 0.000,B 0.000,C 180.000,E1 0.000} C_DIS
LIN {X -173.970,Y 187.955,Z 100.000,A 0.000,B 0.000,C 180.000,E1 0.000} C_DIS
LIN {X -183.414,Y 178.752,Z 100.000,A 0.000,B 0.000,C 180.000,E1 0.000} C_DIS
LIN {X -192.373,Y 169.072,Z 100.000,A 0.000,B 0.000,C 180.000,E1 0.000} C_DIS
LIN {X -200.821,Y 158.944,Z 100.000,A 0.000,B 0.000,C 180.000,E1 0.000} C_DIS
LIN {X -208.738,Y 148.396,Z 100.000,A 0.000,B 0.000,C 180.000,E1 0.000} C_DIS
LIN {X -216.101,Y 137.453,Z 100.000,A 0.000,B 0.000,C 180.000,E1 0.000} C_DIS
LIN {X -222.890,Y 126.147,Z 100.000,A 0.000,B 0.000,C 180.000,E1 0.000} C_DIS
LIN {X -229.088,Y 114.506,Z 100.000,A 0.000,B 0.000,C 180.000,E1 0.000} C_DIS
LIN {X -234.678,Y 102.560,Z 100.000,A 0.000,B 0.000,C 180.000,E1 0.000} C_DIS
LIN {X -239.647,Y 90.343,Z 100.000,A 0.000,B 0.000,C 180.000,E1 0.000} C_DIS
LIN {X -243.981,Y 77.886,Z 100.000,A 0.000,B 0.000,C 180.000,E1 0.000} C_DIS
LIN {X -247.667,Y 65.225,Z 100.000,A 0.000,B 0.000,C 180.000,E1 0.000} C_DIS
LIN {X -250.695,Y 52.389,Z 100.000,A 0.000,B 0.000,C 180.000,E1 0.000} C_DIS
LIN {X -253.060,Y 39.412,Z 100.000,A 0.000,B 0.000,C 180.000,E1 0.000} C_DIS
LIN {X -254.753,Y 26.333,Z 100.000,A 0.000,B 0.000,C 180.000,E1 0.000} C_DIS
LIN {X -255.772,Y 13.184,Z 100.000,A 0.000,B 0.000,C 180.000,E1 0.000} C_DIS
LIN {X -256.111,Y 0.000,Z 100.000,A 0.000,B 0.000,C 180.000,E1 0.000} C_DIS
LIN {X -255.772,Y -13.184,Z 100.000,A 0.000,B 0.000,C 180.000,E1 0.000} C_DIS
LIN {X -254.753,Y -26.333,Z 100.000,A 0.000,B 0.000,C 180.000,E1 0.000} C_DIS
LIN {X -253.060,Y -39.412,Z 100.000,A 0.000,B 0.000,C 180.000,E1 0.000} C_DIS
LIN {X -250.695,Y -52.389,Z 100.000,A 0.000,B 0.000,C 180.000,E1 0.000} C_DIS
LIN {X -247.667,Y -65.225,Z 100.000,A 0.000,B 0.000,C 180.000,E1 0.000} C_DIS
LIN {X -243.981,Y -77.886,Z 100.000,A 0.000,B 0.000,C 180.000,E1 0.000} C_DIS
LIN {X -239.647,Y -90.343,Z 100.000,A 0.000,B 0.000,C 180.000,E1 0.000} C_DIS
LIN {X -234.678,Y -102.560,Z 100.000,A 0.000,B 0.000,C 180.000,E1 0.000} C_DIS
LIN {X -229.088,Y -114.506,Z 100.000,A 0.000,B 0.000,C 180.000,E1 0.000} C_DIS
LIN {X -222.890,Y -126.146,Z 100.000,A 0.000,B 0.000,C 180.000,E1 0.000} C_DIS
LIN {X -216.100,Y -137.454,Z 100.000,A 0.000,B 0.000,C 180.000,E1 0.000} C_DIS
LIN {X -208.738,Y -148.396,Z 100.000,A 0.000,B 0.000,C 180.000,E1 0.000} C_DIS
LIN {X -200.821,Y -158.944,Z 100.000,A 0.000,B 0.000,C 180.000,E1 0.000} C_DIS
LIN {X -192.373,Y -169.072,Z 100.000,A 0.000,B 0.000,C 180.000,E1 0.000} C_DIS
LIN {X -183.414,Y -178.752,Z 100.000,A 0.000,B 0.000,C 180.000,E1 0.000} C_DIS
LIN {X -173.970,Y -187.955,Z 100.000,A 0.000,B 0.000,C 180.000,E1 0.000} C_DIS
LIN {X -164.063,Y -196.662,Z 100.000,A 0.000,B 0.000,C 180.000,E1 0.000} C_DIS
LIN {X -153.721,Y -204.847,Z 100.000,A 0.000,B 0.000,C 180.000,E1 0.000} C_DIS
LIN {X -142.972,Y -212.489,Z 100.000,A 0.000,B 0.000,C 180.000,E1 0.000} C_DIS
LIN {X -131.844,Y -219.568,Z 100.000,A 0.000,B 0.000,C 180.000,E1 0.000} C_DIS
LIN {X -120.365,Y -226.064,Z 100.000,A 0.000,B 0.000,C 180.000,E1 0.000} C_DIS
LIN {X -108.569,Y -231.960,Z 100.000,A 0.000,B 0.000,C 180.000,E1 0.000} C_DIS
LIN {X -96.484,Y -237.241,Z 100.000,A 0.000,B 0.000,C 180.000,E1 0.000} C_DIS
LIN {X -84.142,Y -241.894,Z 100.000,A 0.000,B 0.000,C 180.000,E1 0.000} C_DIS
LIN {X -71.579,Y -245.905,Z 100.000,A 0.000,B 0.000,C 180.000,E1 0.000} C_DIS
LIN {X -58.826,Y -249.263,Z 100.000,A 0.000,B 0.000,C 180.000,E1 0.000} C_DIS
LIN {X -45.916,Y -251.961,Z 100.000,A 0.000,B 0.000,C 180.000,E1 0.000} C_DIS
LIN {X -32.884,Y -253.991,Z 100.000,A 0.000,B 0.000,C 180.000,E1 0.000} C_DIS
LIN {X -19.765,Y -255.347,Z 100.000,A 0.000,B 0.000,C 180.000,E1 0.000} C_DIS
LIN {X -6.594,Y -256.026,Z 100.000,A 0.000,B 0.000,C 180.000,E1 0.000} C_DIS
LIN {X 6.595,Y -256.026,Z 100.000,A 0.000,B 0.000,C 180.000,E1 0.000} C_DIS
LIN {X 16.157,Y -255.533,Z 100.000,A 0.000,B 0.000,C 180.000,E1 0.000} C_DIS
LIN {X 19.764,Y -255.347,Z 100.000,A 0.000,B 0.000,C 180.000,E1 0.000} C_DIS
LIN {X 32.884,Y -253.991,Z 100.000,A 0.000,B 0.000,C 180.000,E1 0.000} C_DIS
LIN {X 45.916,Y -251.961,Z 100.000,A 0.000,B 0.000,C 180.000,E1 0.000} C_DIS
LIN {X 58.826,Y -249.263,Z 100.000,A 0.000,B 0.000,C 180.000,E1 0.000} C_DIS
LIN {X 71.579,Y -245.905,Z 100.000,A 0.000,B 0.000,C 180.000,E1 0.000} C_DIS
LIN {X 84.142,Y -241.894,Z 100.000,A 0.000,B 0.000,C 180.000,E1 0.000} C_DIS
LIN {X 96.484,Y -237.241,Z 100.000,A 0.000,B 0.000,C 180.000,E1 0.000} C_DIS
LIN {X 108.569,Y -231.960,Z 100.000,A 0.000,B 0.000,C 180.000,E1 0.000} C_DIS
LIN {X 120.365,Y -226.064,Z 100.000,A 0.000,B 0.000,C 180.000,E1 0.000} C_DIS
LIN {X 131.844,Y -219.568,Z 100.000,A 0.000,B 0.000,C 180.000,E1 0.000} C_DIS
LIN {X 142.972,Y -212.489,Z 100.000,A 0.000,B 0.000,C 180.000,E1 0.000} C_DIS
LIN {X 153.721,Y -204.847,Z 100.000,A 0.000,B 0.000,C 180.000,E1 0.000} C_DIS
LIN {X 164.063,Y -196.662,Z 100.000,A 0.000,B 0.000,C 180.000,E1 0.000} C_DIS
LIN {X 173.970,Y -187.955,Z 100.000,A 0.000,B 0.000,C 180.000,E1 0.000} C_DIS
LIN {X 183.414,Y -178.752,Z 100.000,A 0.000,B 0.000,C 180.000,E1 0.000} C_DIS
LIN {X 192.373,Y -169.072,Z 100.000,A 0.000,B 0.000,C 180.000,E1 0.000} C_DIS
LIN {X 200.821,Y -158.944,Z 100.000,A 0.000,B 0.000,C 180.000,E1 0.000} C_DIS
LIN {X 208.738,Y -148.396,Z 100.000,A 0.000,B 0.000,C 180.000,E1 0.000} C_DIS
LIN {X 216.101,Y -137.453,Z 100.000,A 0.000,B 0.000,C 180.000,E1 0.000} C_DIS
LIN {X 222.890,Y -126.147,Z 100.000,A 0.000,B 0.000,C 180.000,E1 0.000} C_DIS
LIN {X 229.088,Y -114.506,Z 100.000,A 0.000,B 0.000,C 180.000,E1 0.000} C_DIS
LIN {X 234.678,Y -102.560,Z 100.000,A 0.000,B 0.000,C 180.000,E1 0.000} C_DIS
LIN {X 239.647,Y -90.343,Z 100.000,A 0.000,B 0.000,C 180.000,E1 0.000} C_DIS
LIN {X 243.981,Y -77.886,Z 100.000,A 0.000,B 0.000,C 180.000,E1 0.000} C_DIS
LIN {X 247.667,Y -65.225,Z 100.000,A 0.000,B 0.000,C 180.000,E1 0.000} C_DIS
LIN {X 250.695,Y -52.389,Z 100.000,A 0.000,B 0.000,C 180.000,E1 0.000} C_DIS
LIN {X 253.060,Y -39.412,Z 100.000,A 0.000,B 0.000,C 180.000,E1 0.000} C_DIS
LIN {X 254.753,Y -26.333,Z 100.000,A 0.000,B 0.000,C 180.000,E1 0.000} C_DIS
LIN {X 255.772,Y -13.184,Z 100.000,A 0.000,B 0.000,C 180.000,E1 0.000} C_DIS
LIN {X 256.111,Y 0.000,Z 100.000,A 0.000,B 0.000,C 180.000,E1 0.000} C_DIS
LIN {X 255.772,Y 13.184,Z 100.000,A 0.000,B 0.000,C 180.000,E1 0.000} C_DIS
LIN {X 254.753,Y 26.333,Z 100.000,A 0.000,B 0.000,C 180.000,E1 0.000} C_DIS
LIN {X 253.060,Y 39.412,Z 100.000,A 0.000,B 0.000,C 180.000,E1 0.000} C_DIS
LIN {X 250.695,Y 52.389,Z 100.000,A 0.000,B 0.000,C 180.000,E1 0.000} C_DIS
LIN {X 247.667,Y 65.225,Z 100.000,A 0.000,B 0.000,C 180.000,E1 0.000} C_DIS
LIN {X 243.981,Y 77.886,Z 100.000,A 0.000,B 0.000,C 180.000,E1 0.000} C_DIS
LIN {X 239.647,Y 90.343,Z 100.000,A 0.000,B 0.000,C 180.000,E1 0.000} C_DIS
LIN {X 234.678,Y 102.560,Z 100.000,A 0.000,B 0.000,C 180.000,E1 0.000} C_DIS
LIN {X 229.088,Y 114.506,Z 100.000,A 0.000,B 0.000,C 180.000,E1 0.000} C_DIS
LIN {X 222.890,Y 126.146,Z 100.000,A 0.000,B 0.000,C 180.000,E1 0.000} C_DIS
LIN {X 216.100,Y 137.454,Z 100.000,A 0.000,B 0.000,C 180.000,E1 0.000} C_DIS
LIN {X 208.738,Y 148.396,Z 100.000,A 0.000,B 0.000,C 180.000,E1 0.000} C_DIS
LIN {X 200.821,Y 158.944,Z 100.000,A 0.000,B 0.000,C 180.000,E1 0.000} C_DIS
LIN {X 192.373,Y 169.072,Z 100.000,A 0.000,B 0.000,C 180.000,E1 0.000} C_DIS
LIN {X 183.414,Y 178.752,Z 100.000,A 0.000,B 0.000,C 180.000,E1 0.000} C_DIS
LIN {X 173.970,Y 187.955,Z 100.000,A 0.000,B 0.000,C 180.000,E1 0.000} C_DIS
LIN {X 164.063,Y 196.662,Z 100.000,A 0.000,B 0.000,C 180.000,E1 0.000} C_DIS
LIN {X 153.721,Y 204.847,Z 100.000,A 0.000,B 0.000,C 180.000,E1 0.000} C_DIS
LIN {X 142.972,Y 212.489,Z 100.000,A 0.000,B 0.000,C 180.000,E1 0.000} C_DIS
;rapid-leaky
$VEL.CP=0.3
LIN {X 49.451,Y -233.079,Z 100.000,A 0.000,B 0.000,C 180.000,E1 0.000} C_DIS
;bead-sparse_infill
$VEL.CP=0.68
LIN {X 233.159,Y -49.370,Z 100.000,A 0.000,B 0.000,C 180.000,E1 0.000} C_DIS
LIN {X 233.304,Y -48.755,Z 100.000,A 0.000,B 0.000,C 180.000,E1 0.000} C_DIS
LIN {X 235.506,Y -36.678,Z 100.000,A 0.000,B 0.000,C 180.000,E1 0.000} C_DIS
LIN {X 237.082,Y -24.506,Z 100.000,A 0.000,B 0.000,C 180.000,E1 0.000} C_DIS
LIN {X 238.029,Y -12.269,Z 100.000,A 0.000,B 0.000,C 180.000,E1 0.000} C_DIS
LIN {X 238.345,Y 0.000,Z 100.000,A 0.000,B 0.000,C 180.000,E1 0.000} C_DIS
LIN {X 238.029,Y 12.269,Z 100.000,A 0.000,B 0.000,C 180.000,E1 0.000} C_DIS
LIN {X 237.082,Y 24.506,Z 100.000,A 0.000,B 0.000,C 180.000,E1 0.000} C_DIS
LIN {X 235.506,Y 36.678,Z 100.000,A 0.000,B 0.000,C 180.000,E1 0.000} C_DIS
LIN {X 233.304,Y 48.755,Z 100.000,A 0.000,B 0.000,C 180.000,E1 0.000} C_DIS
LIN {X 230.486,Y 60.701,Z 100.000,A 0.000,B 0.000,C 180.000,E1 0.000} C_DIS
LIN {X 227.056,Y 72.483,Z 100.000,A 0.000,B 0.000,C 180.000,E1 0.000} C_DIS
LIN {X 223.024,Y 84.076,Z 100.000,A 0.000,B 0.000,C 180.000,E1 0.000} C_DIS
LIN {X 219.150,Y 93.599,Z 100.000,A 0.000,B 0.000,C 180.000,E1 0.000} C_DIS
LIN {X -93.578,Y -219.130,Z 100.000,A 0.000,B 0.000,C 180.000,E1 0.000} C_DIS
LIN {X -101.038,Y -215.869,Z 100.000,A 0.000,B 0.000,C 180.000,E1 0.000} C_DIS
LIN {X -112.016,Y -210.382,Z 100.000,A 0.000,B 0.000,C 180.000,E1 0.000} C_DIS
LIN {X -122.698,Y -204.337,Z 100.000,A 0.000,B 0.000,C 180.000,E1 0.000} C_DIS
LIN {X -133.055,Y -197.749,Z 100.000,A 0.000,B 0.000,C 180.000,E1 0.000} C_DIS
LIN {X -143.057,Y -190.638,Z 100.000,A 0.000,B 0.000,C 180.000,E1 0.000} C_DIS
LIN {X -152.682,Y -183.020,Z 100.000,A 0.000,B 0.000,C 180.000,E1 0.000} C_DIS
LIN {X -161.902,Y -174.917,Z 100.000,A 0.000,B 0.000,C 180.000,E1 0.000} C_DIS
LIN {X -170.691,Y -166.352,Z 100.000,A 0.000,B 0.000,C 180.000,E1 0.000} C_DIS
LIN {X -179.028,Y -157.345,Z 100.000,A 0.000,B 0.000,C 180.000,E1 0.000} C_DIS
LIN {X -183.459,Y -152.033,Z 100.000,A 0.000,B 0.000,C 180.000,E1 0.000} C_DIS
LIN {X 152.075,Y 183.501,Z 100.000,A 0.000,B 0.000,C 180.000,E1 0.000} C_DIS
LIN {X 143.057,Y 190.638,Z 100.000,A 0.000,B 0.000,C 180.000,E1 0.000} C_DIS
LIN {X 133.055,Y 197.749,Z 100.000,A 0.000,B 0.000,C 180.000,E1 0.000} C_DIS
LIN {X 122.698,Y 204.337,Z 100.000,A 0.000,B 0.000,C 180.000,E1 0.000} C_DIS
LIN {X 112.016,Y 210.382,Z 100.000,A 0.000,B 0.000,C 180.000,E1 0.000} C_DIS
LIN {X 101.038,Y 215.869,Z 100.000,A 0.000,B 0.000,C 180.000,E1 0.000} C_DIS
LIN {X 89.792,Y 220.784,Z 100.000,A 0.000,B 0.000,C 180.000,E1 0.000} C_DIS
LIN {X 78.305,Y 225.114,Z 100.000,A 0.000,B 0.000,C 180.000,E1 0.000} C_DIS
LIN {X 66.613,Y 228.847,Z 100.000,A 0.000,B 0.000,C 180.000,E1 0.000} C_DIS
LIN {X 54.746,Y 231.972,Z 100.000,A 0.000,B 0.000,C 180.000,E1 0.000} C_DIS
LIN {X 45.500,Y 233.904,Z 100.000,A 0.000,B 0.000,C 180.000,E1 0.000} C_DIS
LIN {X -233.898,Y -45.495,Z 100.000,A 0.000,B 0.000,C 180.000,E1 0.000} C_DIS
;rapid-leaky
$VEL.CP=0.3
LIN {X -149.554,Y 222.273,Z 110.000,A 0.000,B 0.000,C 180.000,E1 0.000} C_DIS
;bead-perimeter_outer
$VEL.CP=0.68
LIN {X -160.799,Y 214.279,Z 110.000,A 0.000,B 0.000,C 180.000,E1 0.000} C_DIS
LIN {X -171.616,Y 205.717,Z 110.000,A 0.000,B 0.000,C 180.000,E1 0.000} C_DIS
LIN {X -181.980,Y 196.610,Z 110.000,A 0.000,B 0.000,C 180.000,E1 0.000} C_DIS
LIN {X -191.859,Y 186.981,Z 110.000,A 0.000,B 0.000,C 180.000,E1 0.000} C_DIS
LIN {X -195.633,Y 182.905,Z 110.000,A 0.000,B 0.000,C 180.000,E1 0.000} C_DIS
LIN {X -201.230,Y 176.857,Z 110.000,A 0.000,B 0.000,C 180.000,E1 0.000} C_DIS
LIN {X -210.067,Y 166.263,Z 110.000,A 0.000,B 0.000,C 180.000,E1 0.000} C_DIS
LIN {X -218.348,Y 155.228,Z 110.000,A 0.000,B 0.000,C 180.000,E1 0.000} C_DIS
LIN {X -226.050,Y 143.781,Z 110.000,A 0.000,B 0.000,C 180.000,E1 0.000} C_DIS
LIN {X -233.153,Y 131.955,Z 110.000,A 0.000,B 0.000,C 180.000,E1 0.000} C_DIS
LIN {X -239.636,Y 119.778,Z 110.000,A 0.000,B 0.000,C 180.000,E1 0.000} C_DIS
LIN {X -245.483,Y 107.283,Z 110.000,A 0.000,B 0.000,C 180.000,E1 0.000} C_DIS
LIN {X -250.681,Y 94.503,Z 110.000,A 0.000,B 0.000,C 180.000,E1 0.000} C_DIS
LIN {X -255.214,Y 81.473,Z 110.000,A 0.000,B 0.000,C 180.000,E1 0.000} C_DIS
LIN {X -259.069,Y 68.227,Z 110.000,A 0.000,B 0.000,C 180.000,E1 0.000} C_DIS
LIN {X -262.238,Y 54.800,Z 110.000,A 0.000,B 0.000,C 180.000,E1 0.000} C_DIS
LIN {X -264.711,Y 41.227,Z 110.000,A 0.000,B 0.000,C 180.000,E1 0.000} C_DIS
LIN {X -266.483,Y 27.545,Z 110.000,A 0.000,B 0.000,C 180.000,E1 0.000} C_DIS
LIN {X -267.548,Y 13.792,Z 110.000,A 0.000,B 0.000,C 180.000,E1 0.000} C_DIS
LIN {X -267.902,Y 0.000,Z 110.000,A 0.000,B 0.000,C 180.000,E1 0.000} C_DIS
LIN {X -267.548,Y -13.792,Z 110.000,A 0.000,B 0.000,C 180.000,E1 0.000} C_DIS
LIN {X -266.483,Y -27.545,Z 110.000,A 0.000,B 0.000,C 180.000,E1 0.000} C_DIS
LIN {X -264.711,Y -41.227,Z 110.000,A 0.000,B 0.000,C 180.000,E1 0.000} C_DIS
LIN {X -262.238,Y -54.800,Z 110.000,A 0.000,B 0.000,C 180.000,E1 0.000} C_DIS
LIN {X -259.069,Y -68.227,Z 110.000,A 0.000,B 0.000,C 180.000,E1 0.000} C_DIS
LIN {X -255.214,Y -81.473,Z 110.000,A 0.000,B 0.000,C 180.000,E1 0.000} C_DIS
LIN {X -250.681,Y -94.503,Z 110.000,A 0.000,B 0.000,C 180.000,E1 0.000} C_DIS
LIN {X -245.483,Y -107.283,Z 110.000,A 0.000,B 0.000,C 180.000,E1 0.000} C_DIS
LIN {X -239.636,Y -119.778,Z 110.000,A 0.000,B 0.000,C 180.000,E1 0.000} C_DIS
LIN {X -233.153,Y -131.955,Z 110.000,A 0.000,B 0.000,C 180.000,E1 0.000} C_DIS
LIN {X -226.050,Y -143.781,Z 110.000,A 0.000,B 0.000,C 180.000,E1 0.000} C_DIS
LIN {X -218.348,Y -155.228,Z 110.000,A 0.000,B 0.000,C 180.000,E1 0.000} C_DIS
LIN {X -210.067,Y -166.263,Z 110.000,A 0.000,B 0.000,C 180.000,E1 0.000} C_DIS
LIN {X -201.231,Y -176.857,Z 110.000,A 0.000,B 0.000,C 180.000,E1 0.000} C_DIS
LIN {X -191.859,Y -186.981,Z 110.000,A 0.000,B 0.000,C 180.000,E1 0.000} C_DIS
LIN {X -181.980,Y -196.610,Z 110.000,A 0.000,B 0.000,C 180.000,E1 0.000} C_DIS
LIN {X -171.616,Y -205.717,Z 110.000,A 0.000,B 0.000,C 180.000,E1 0.000} C_DIS
LIN {X -160.799,Y -214.279,Z 110.000,A 0.000,B 0.000,C 180.000,E1 0.000} C_DIS
LIN {X -149.554,Y -222.273,Z 110.000,A 0.000,B 0.000,C 180.000,E1 0.000} C_DIS
LIN {X -137.914,Y -229.678,Z 110.000,A 0.000,B 0.000,C 180.000,E1 0.000} C_DIS
LIN {X -125.908,Y -236.472,Z 110.000,A 0.000,B 0.000,C 180.000,E1 0.000} C_DIS
LIN {X -113.568,Y -242.640,Z 110.000,A 0.000,B 0.000,C 180.000,E1 0.000} C_DIS
LIN {X -100.926,Y -248.165,Z 110.000,A 0.000,B 0.000,C 180.000,E1 0.000} C_DIS
LIN {X -88.017,Y -253.032,Z 110.000,A 0.000,B 0.000,C 180.000,E1 0.000} C_DIS
LIN {X -74.875,Y -257.227,Z 110.000,A 0.000,B 0.000,C 180.000,E1 0.000} C_DIS
LIN {X -61.534,Y -260.740,Z 110.000,A 0.000,B 0.000,C 180.000,E1 0.000} C_DIS
LIN {X -48.029,Y -263.562,Z 110.000,A 0.000,B 0.000,C 180.000,E1 0.000} C_DIS
LIN {X -34.398,Y -265.685,Z 110.000,A 0.000,B 0.000,C 180.000,E1 0.000} C_DIS
LIN {X -20.675,Y -267.103,Z 110.000,A 0.000,B 0.000,C 180.000,E1 0.000} C_DIS
LIN {X -6.898,Y -267.814,Z 110.000,A 0.000,B 0.000,C 180.000,E1 0.000} C_DIS
LIN {X 6.898,Y -267.814,Z 110.000,A 0.000,B 0.000,C 180.000,E1 0.000} C_DIS
LIN {X 20.675,Y -267.103,Z 110.000,A 0.000,B 0.000,C 180.000,E1 0.000} C_DIS
LIN {X 34.398,Y -265.685,Z 110.000,A 0.000,B 0.000,C 180.000,E1 0.000} C_DIS
LIN {X 48.029,Y -263.562,Z 110.000,A 0.000,B 0.000,C 180.000,E1 0.000} C_DIS
LIN {X 61.534,Y -260.740,Z 110.000,A 0.000,B 0.000,C 180.000,E1 0.000} C_DIS
LIN {X 74.875,Y -257.227,Z 110.000,A 0.000,B 0.000,C 180.000,E1 0.000} C_DIS
LIN {X 88.017,Y -253.032,Z 110.000,A 0.000,B 0.000,C 180.000,E1 0.000} C_DIS
LIN {X 100.926,Y -248.165,Z 110.000,A 0.000,B 0.000,C 180.000,E1 0.000} C_DIS
LIN {X 113.568,Y -242.640,Z 110.000,A 0.000,B 0.000,C 180.000,E1 0.000} C_DIS
LIN {X 125.908,Y -236.472,Z 110.000,A 0.000,B 0.000,C 180.000,E1 0.000} C_DIS
LIN {X 137.914,Y -229.678,Z 110.000,A 0.000,B 0.000,C 180.000,E1 0.000} C_DIS
LIN {X 149.554,Y -222.273,Z 110.000,A 0.000,B 0.000,C 180.000,E1 0.000} C_DIS
LIN {X 160.799,Y -214.279,Z 110.000,A 0.000,B 0.000,C 180.000,E1 0.000} C_DIS
LIN {X 171.616,Y -205.717,Z 110.000,A 0.000,B 0.000,C 180.000,E1 0.000} C_DIS
LIN {X 181.980,Y -196.610,Z 110.000,A 0.000,B 0.000,C 180.000,E1 0.000} C_DIS
LIN {X 191.859,Y -186.981,Z 110.000,A 0.000,B 0.000,C 180.000,E1 0.000} C_DIS
LIN {X 195.632,Y -182.906,Z 110.000,A 0.000,B 0.000,C 180.000,E1 0.000} C_DIS
LIN {X 201.230,Y -176.857,Z 110.000,A 0.000,B 0.000,C 180.000,E1 0.000} C_DIS
LIN {X 210.067,Y -166.263,Z 110.000,A 0.000,B 0.000,C 180.000,E1 0.000} C_DIS
LIN {X 218.348,Y -155.228,Z 110.000,A 0.000,B 0.000,C 180.000,E1 0.000} C_DIS
LIN {X 226.050,Y -143.781,Z 110.000,A 0.000,B 0.000,C 180.000,E1 0.000} C_DIS
LIN {X 233.153,Y -131.955,Z 110.000,A 0.000,B 0.000,C 180.000,E1 0.000} C_DIS
LIN {X 239.636,Y -119.778,Z 110.000,A 0.000,B 0.000,C 180.000,E1 0.000} C_DIS
LIN {X 245.483,Y -107.283,Z 110.000,A 0.000,B 0.000,C 180.000,E1 0.000} C_DIS
LIN {X 250.681,Y -94.503,Z 110.000,A 0.000,B 0.000,C 180.000,E1 0.000} C_DIS
LIN {X 255.214,Y -81.473,Z 110.000,A 0.000,B 0.000,C 180.000,E1 0.000} C_DIS
LIN {X 259.069,Y -68.227,Z 110.000,A 0.000,B 0.000,C 180.000,E1 0.000} C_DIS
LIN {X 262.238,Y -54.800,Z 110.000,A 0.000,B 0.000,C 180.000,E1 0.000} C_DIS
LIN {X 264.711,Y -41.227,Z 110.000,A 0.000,B 0.000,C 180.000,E1 0.000} C_DIS
LIN {X 266.483,Y -27.545,Z 110.000,A 0.000,B 0.000,C 180.000,E1 0.000} C_DIS
LIN {X 267.548,Y -13.792,Z 110.000,A 0.000,B 0.000,C 180.000,E1 0.000} C_DIS
LIN {X 267.902,Y 0.000,Z 110.000,A 0.000,B 0.000,C 180.000,E1 0.000} C_DIS
LIN {X 267.548,Y 13.792,Z 110.000,A 0.000,B 0.000,C 180.000,E1 0.000} C_DIS
LIN {X 266.483,Y 27.545,Z 110.000,A 0.000,B 0.000,C 180.000,E1 0.000} C_DIS
LIN {X 264.711,Y 41.227,Z 110.000,A 0.000,B 0.000,C 180.000,E1 0.000} C_DIS
LIN {X 262.238,Y 54.800,Z 110.000,A 0.000,B 0.000,C 180.000,E1 0.000} C_DIS
LIN {X 259.069,Y 68.227,Z 110.000,A 0.000,B 0.000,C 180.000,E1 0.000} C_DIS
LIN {X 255.214,Y 81.473,Z 110.000,A 0.000,B 0.000,C 180.000,E1 0.000} C_DIS
LIN {X 250.681,Y 94.503,Z 110.000,A 0.000,B 0.000,C 180.000,E1 0.000} C_DIS
LIN {X 245.483,Y 107.283,Z 110.000,A 0.000,B 0.000,C 180.000,E1 0.000} C_DIS
LIN {X 239.636,Y 119.778,Z 110.000,A 0.000,B 0.000,C 180.000,E1 0.000} C_DIS
LIN {X 233.153,Y 131.955,Z 110.000,A 0.000,B 0.000,C 180.000,E1 0.000} C_DIS
LIN {X 226.050,Y 143.781,Z 110.000,A 0.000,B 0.000,C 180.000,E1 0.000} C_DIS
LIN {X 218.348,Y 155.228,Z 110.000,A 0.000,B 0.000,C 180.000,E1 0.000} C_DIS
LIN {X 215.015,Y 159.670,Z 110.000,A 0.000,B 0.000,C 180.000,E1 0.000} C_DIS
LIN {X 210.067,Y 166.263,Z 110.000,A 0.000,B 0.000,C 180.000,E1 0.000} C_DIS
LIN {X 201.231,Y 176.857,Z 110.000,A 0.000,B 0.000,C 180.000,E1 0.000} C_DIS
LIN {X 191.859,Y 186.981,Z 110.000,A 0.000,B 0.000,C 180.000,E1 0.000} C_DIS
LIN {X 181.980,Y 196.610,Z 110.000,A 0.000,B 0.000,C 180.000,E1 0.000} C_DIS
LIN {X 171.616,Y 205.717,Z 110.000,A 0.000,B 0.000,C 180.000,E1 0.000} C_DIS
LIN {X 160.799,Y 214.279,Z 110.000,A 0.000,B 0.000,C 180.000,E1 0.000} C_DIS
LIN {X 149.554,Y 222.273,Z 110.000,A 0.000,B 0.000,C 180.000,E1 0.000} C_DIS
LIN {X 137.914,Y 229.678,Z 110.000,A 0.000,B 0.000,C 180.000,E1 0.000} C_DIS
LIN {X 125.908,Y 236.472,Z 110.000,A 0.000,B 0.000,C 180.000,E1 0.000} C_DIS
LIN {X 113.568,Y 242.640,Z 110.000,A 0.000,B 0.000,C 180.000,E1 0.000} C_DIS
LIN {X 100.926,Y 248.165,Z 110.000,A 0.000,B 0.000,C 180.000,E1 0.000} C_DIS
LIN {X 88.017,Y 253.032,Z 110.000,A 0.000,B 0.000,C 180.000,E1 0.000} C_DIS
LIN {X 74.875,Y 257.227,Z 110.000,A 0.000,B 0.000,C 180.000,E1 0.000} C_DIS
LIN {X 61.534,Y 260.740,Z 110.000,A 0.000,B 0.000,C 180.000,E1 0.000} C_DIS
LIN {X 48.029,Y 263.562,Z 110.000,A 0.000,B 0.000,C 180.000,E1 0.000} C_DIS
LIN {X 34.398,Y 265.685,Z 110.000,A 0.000,B 0.000,C 180.000,E1 0.000} C_DIS
LIN {X 20.675,Y 267.103,Z 110.000,A 0.000,B 0.000,C 180.000,E1 0.000} C_DIS
LIN {X 6.898,Y 267.814,Z 110.000,A 0.000,B 0.000,C 180.000,E1 0.000} C_DIS
LIN {X -6.898,Y 267.814,Z 110.000,A 0.000,B 0.000,C 180.000,E1 0.000} C_DIS
LIN {X -20.675,Y 267.103,Z 110.000,A 0.000,B 0.000,C 180.000,E1 0.000} C_DIS
LIN {X -34.398,Y 265.685,Z 110.000,A 0.000,B 0.000,C 180.000,E1 0.000} C_DIS
LIN {X -48.029,Y 263.562,Z 110.000,A 0.000,B 0.000,C 180.000,E1 0.000} C_DIS
LIN {X -61.534,Y 260.740,Z 110.000,A 0.000,B 0.000,C 180.000,E1 0.000} C_DIS
LIN {X -74.875,Y 257.227,Z 110.000,A 0.000,B 0.000,C 180.000,E1 0.000} C_DIS
LIN {X -88.017,Y 253.032,Z 110.000,A 0.000,B 0.000,C 180.000,E1 0.000} C_DIS
LIN {X -100.926,Y 248.165,Z 110.000,A 0.000,B 0.000,C 180.000,E1 0.000} C_DIS
LIN {X -113.568,Y 242.640,Z 110.000,A 0.000,B 0.000,C 180.000,E1 0.000} C_DIS
LIN {X -125.908,Y 236.472,Z 110.000,A 0.000,B 0.000,C 180.000,E1 0.000} C_DIS
LIN {X -137.914,Y 229.678,Z 110.000,A 0.000,B 0.000,C 180.000,E1 0.000} C_DIS
LIN {X -149.554,Y 222.273,Z 110.000,A 0.000,B 0.000,C 180.000,E1 0.000} C_DIS
;rapid-leaky
$VEL.CP=0.3
LIN {X -140.876,Y 209.375,Z 110.000,A 0.000,B 0.000,C 180.000,E1 0.000} C_DIS
;bead-perimeter_inner
$VEL.CP=0.68
LIN {X -151.469,Y 201.845,Z 110.000,A 0.000,B 0.000,C 180.000,E1 0.000} C_DIS
LIN {X -161.658,Y 193.780,Z 110.000,A 0.000,B 0.000,C 180.000,E1 0.000} C_DIS
LIN {X -171.421,Y 185.201,Z 110.000,A 0.000,B 0.000,C 180.000,E1 0.000} C_DIS
LIN {X -180.727,Y 176.131,Z 110.000,A 0.000,B 0.000,C 180.000,E1 0.000} C_DIS
LIN {X -189.553,Y 166.596,Z 110.000,A 0.000,B 0.000,C 180.000,E1 0.000} C_DIS
LIN {X -197.878,Y 156.616,Z 110.000,A 0.000,B 0.000,C 180.000,E1 0.000} C_DIS
LIN {X -205.679,Y 146.221,Z 110.000,A 0.000,B 0.000,C 180.000,E1 0.000} C_DIS
LIN {X -212.934,Y 135.438,Z 110.000,A 0.000,B 0.000,C 180.000,E1 0.000} C_DIS
LIN {X -219.624,Y 124.298,Z 110.000,A 0.000,B 0.000,C 180.000,E1 0.000} C_DIS
LIN {X -225.731,Y 112.828,Z 110.000,A 0.000,B 0.000,C 180.000,E1 0.000} C_DIS
LIN {X -231.239,Y 101.058,Z 110.000,A 0.000,B 0.000,C 180.000,E1 0.000} C_DIS
LIN {X -236.136,Y 89.019,Z 110.000,A 0.000,B 0.000,C 180.000,E1 0.000} C_DIS
LIN {X -240.405,Y 76.746,Z 110.000,A 0.000,B 0.000,C 180.000,E1 0.000} C_DIS
LIN {X -244.037,Y 64.269,Z 110.000,A 0.000,B 0.000,C 180.000,E1 0.000} C_DIS
LIN {X -247.021,Y 51.621,Z 110.000,A 0.000,B 0.000,C 180.000,E1 0.000} C_DIS
LIN {X -249.351,Y 38.835,Z 110.000,A 0.000,B 0.000,C 180.000,E1 0.000} C_DIS
LIN {X -251.021,Y 25.946,Z 110.000,A 0.000,B 0.000,C 180.000,E1 0.000} C_DIS
LIN {X -252.023,Y 12.992,Z 110.000,A 0.000,B 0.000,C 180.000,E1 0.000} C_DIS
LIN {X -252.357,Y 0.000,Z 110.000,A 0.000,B 0.000,C 180.000,E1 0.000} C_DIS
LIN {X -252.023,Y -12.992,Z 110.000,A 0.000,B 0.000,C 180.000,E1 0.000} C_DIS
LIN {X -251.021,Y -25.946,Z 110.000,A 0.000,B 0.000,C 180.000,E1 0.000} C_DIS
LIN {X -249.351,Y -38.835,Z 110.000,A 0.000,B 0.000,C 180.000,E1 0.000} C_DIS
LIN {X -247.021,Y -51.621,Z 110.000,A 0.000,B 0.000,C 180.000,E1 0.000} C_DIS
LIN {X -244.037,Y -64.269,Z 110.000,A 0.000,B 0.000,C 180.000,E1 0.000} C_DIS
LIN {X -240.405,Y -76.746,Z 110.000,A 0.000,B 0.000,C 180.000,E1 0.000} C_DIS
LIN {X -236.136,Y -89.019,Z 110.000,A 0.000,B 0.000,C 180.000,E1 0.000} C_DIS
LIN {X -231.239,Y -101.058,Z 110.000,A 0.000,B 0.000,C 180.000,E1 0.000} C_DIS
LIN {X -225.731,Y -112.828,Z 110.000,A 0.000,B 0.000,C 180.000,E1 0.000} C_DIS
LIN {X -219.624,Y -124.298,Z 110.000,A 0.000,B 0.000,C 180.000,E1 0.000} C_DIS
LIN {X -212.934,Y -135.438,Z 110.000,A 0.000,B 0.000,C 180.000,E1 0.000} C_DIS
LIN {X -205.678,Y -146.221,Z 110.000,A 0.000,B 0.000,C 180.000,E1 0.000} C_DIS
LIN {X -197.878,Y -156.616,Z 110.000,A 0.000,B 0.000,C 180.000,E1 0.000} C_DIS
LIN {X -189.554,Y -166.595,Z 110.000,A 0.000,B 0.000,C 180.000,E1 0.000} C_DIS
LIN {X -180.726,Y -176.132,Z 110.000,A 0.000,B 0.000,C 180.000,E1 0.000} C_DIS
LIN {X -171.421,Y -185.201,Z 110.000,A 0.000,B 0.000,C 180.000,E1 0.000} C_DIS
LIN {X -161.658,Y -193.780,Z 110.000,A 0.000,B 0.000,C 180.000,E1 0.000} C_DIS
LIN {X -151.469,Y -201.845,Z 110.000,A 0.000,B 0.000,C 180.000,E1 0.000} C_DIS
LIN {X -140.876,Y -209.375,Z 110.000,A 0.000,B 0.000,C 180.000,E1 0.000} C_DIS
LIN {X -129.911,Y -216.351,Z 110.000,A 0.000,B 0.000,C 180.000,E1 0.000} C_DIS
LIN {X -118.602,Y -222.751,Z 110.000,A 0.000,B 0.000,C 180.000,E1 0.000} C_DIS
LIN {X -106.978,Y -228.561,Z 110.000,A 0.000,B 0.000,C 180.000,E1 0.000} C_DIS
LIN {X -95.069,Y -233.766,Z 110.000,A 0.000,B 0.000,C 180.000,E1 0.000} C_DIS
LIN {X -82.911,Y -238.349,Z 110.000,A 0.000,B 0.000,C 180.000,E1 0.000} C_DIS
LIN {X -70.530,Y -242.301,Z 110.000,A 0.000,B 0.000,C 180.000,E1 0.000} C_DIS
LIN {X -57.963,Y -245.611,Z 110.000,A 0.000,B 0.000,C 180.000,E1 0.000} C_DIS
LIN {X -45.242,Y -248.269,Z 110.000,A 0.000,B 0.000,C 180.000,E1 0.000} C_DIS
LIN {X -32.403,Y -250.269,Z 110.000,A 0.000,B 0.000,C 180.000,E1 0.000} C_DIS
LIN {X -19.475,Y -251.605,Z 110.000,A 0.000,B 0.000,C 180.000,E1 0.000} C_DIS
LIN {X -6.497,Y -252.274,Z 110.000,A 0.000,B 0.000,C 180.000,E1 0.000} C_DIS
LIN {X 6.497,Y -252.274,Z 110.000,A 0.000,B 0.000,C 180.000,E1 0.000} C_DIS
LIN {X 19.475,Y -251.605,Z 110.000,A 0.000,B 0.000,C 180.000,E1 0.000} C_DIS
LIN {X 32.403,Y -250.269,Z 110.000,A 0.000,B 0.000,C 180.000,E1 0.000} C_DIS
LIN {X 45.242,Y -248.269,Z 110.000,A 0.000,B 0.000,C 180.000,E1 0.000} C_DIS
LIN {X 57.963,Y -245.611,Z 110.000,A 0.000,B 0.000,C 180.000,E1 0.000} C_DIS
LIN {X 70.530,Y -242.301,Z 110.000,A 0.000,B 0.000,C 180.000,E1 0.000} C_DIS
LIN {X 82.910,Y -238.349,Z 110.000,A 0.000,B 0.000,C 180.000,E1 0.000} C_DIS
LIN {X 95.070,Y -233.766,Z 110.000,A 0.000,B 0.000,C 180.000,E1 0.000} C_DIS
LIN {X 106.978,Y -228.561,Z 110.000,A 0.000,B 0.000,C 180.000,E1 0.000} C_DIS
LIN {X 118.602,Y -222.751,Z 110.000,A 0.000,B 0.000,C 180.000,E1 0.000} C_DIS
LIN {X 129.911,Y -216.351,Z 110.000,A 0.000,B 0.000,C 180.000,E1 0.000} C_DIS
LIN {X 140.876,Y -209.375,Z 110.000,A 0.000,B 0.000,C 180.000,E1 0.000} C_DIS
LIN {X 151.469,Y -201.845,Z 110.000,A 0.000,B 0.000,C 180.000,E1 0.000} C_DIS
LIN {X 161.658,Y -193.780,Z 110.000,A 0.000,B 0.000,C 180.000,E1 0.000} C_DIS
LIN {X 171.421,Y -185.201,Z 110.000,A 0.000,B 0.000,C 180.000,E1 0.000} C_DIS
LIN {X 180.727,Y -176.131,Z 110.000,A 0.000,B 0.000,C 180.000,E1 0.000} C_DIS
LIN {X 189.553,Y -166.596,Z 110.000,A 0.000,B 0.000,C 180.000,E1 0.000} C_DIS
LIN {X 197.878,Y -156.616,Z 110.000,A 0.000,B 0.000,C 180.000,E1 0.000} C_DIS
LIN {X 205.679,Y -146.221,Z 110.000,A 0.000,B 0.000,C 180.000,E1 0.000} C_DIS
LIN {X 212.934,Y -135.438,Z 110.000,A 0.000,B 0.000,C 180.000,E1 0.000} C_DIS
LIN {X 219.624,Y -124.298,Z 110.000,A 0.000,B 0.000,C 180.000,E1 0.000} C_DIS
LIN {X 225.731,Y -112.828,Z 110.000,A 0.000,B 0.000,C 180.000,E1 0.000} C_DIS
LIN {X 231.239,Y -101.058,Z 110.000,A 0.000,B 0.000,C 180.000,E1 0.000} C_DIS
LIN {X 236.136,Y -89.019,Z 110.000,A 0.000,B 0.000,C 180.000,E1 0.000} C_DIS
LIN {X 240.405,Y -76.746,Z 110.000,A 0.000,B 0.000,C 180.000,E1 0.000} C_DIS
LIN {X 244.037,Y -64.269,Z 110.000,A 0.000,B 0.000,C 180.000,E1 0.000} C_DIS
LIN {X 247.021,Y -51.621,Z 110.000,A 0.000,B 0.000,C 180.000,E1 0.000} C_DIS
LIN {X 249.351,Y -38.835,Z 110.000,A 0.000,B 0.000,C 180.000,E1 0.000} C_DIS
LIN {X 251.021,Y -25.946,Z 110.000,A 0.000,B 0.000,C 180.000,E1 0.000} C_DIS
LIN {X 252.023,Y -12.992,Z 110.000,A 0.000,B 0.000,C 180.000,E1 0.000} C_DIS
LIN {X 252.357,Y 0.000,Z 110.000,A 0.000,B 0.000,C 180.000,E1 0.000} C_DIS
LIN {X 252.023,Y 12.992,Z 110.000,A 0.000,B 0.000,C 180.000,E1 0.000} C_DIS
LIN {X 251.021,Y 25.946,Z 110.000,A 0.000,B 0.000,C 180.000,E1 0.000} C_DIS
LIN {X 249.351,Y 38.835,Z 110.000,A 0.000,B 0.000,C 180.000,E1 0.000} C_DIS
LIN {X 247.021,Y 51.621,Z 110.000,A 0.000,B 0.000,C 180.000,E1 0.000} C_DIS
LIN {X 244.037,Y 64.269,Z 110.000,A 0.000,B 0.000,C 180.000,E1 0.000} C_DIS
LIN {X 240.405,Y 76.746,Z 110.000,A 0.000,B 0.000,C 180.000,E1 0.000} C_DIS
LIN {X 236.136,Y 89.019,Z 110.000,A 0.000,B 0.000,C 180.000,E1 0.000} C_DIS
LIN {X 231.239,Y 101.058,Z 110.000,A 0.000,B 0.000,C 180.000,E1 0.000} C_DIS
LIN {X 225.731,Y 112.828,Z 110.000,A 0.000,B 0.000,C 180.000,E1 0.000} C_DIS
LIN {X 219.624,Y 124.298,Z 110.000,A 0.000,B 0.000,C 180.000,E1 0.000} C_DIS
LIN {X 212.934,Y 135.438,Z 110.000,A 0.000,B 0.000,C 180.000,E1 0.000} C_DIS
LIN {X 205.678,Y 146.221,Z 110.000,A 0.000,B 0.000,C 180.000,E1 0.000} C_DIS
LIN {X 197.878,Y 156.616,Z 110.000,A 0.000,B 0.000,C 180.000,E1 0.000} C_DIS
LIN {X 189.554,Y 166.595,Z 110.000,A 0.000,B 0.000,C 180.000,E1 0.000} C_DIS
LIN {X 180.726,Y 176.132,Z 110.000,A 0.000,B 0.000,C 180.000,E1 0.000} C_DIS
LIN {X 171.421,Y 185.201,Z 110.000,A 0.000,B 0.000,C 180.000,E1 0.000} C_DIS
LIN {X 161.658,Y 193.780,Z 110.000,A 0.000,B 0.000,C 180.000,E1 0.000} C_DIS
LIN {X 151.469,Y 201.845,Z 110.000,A 0.000,B 0.000,C 180.000,E1 0.000} C_DIS
LIN {X 140.876,Y 209.375,Z 110.000,A 0.000,B 0.000,C 180.000,E1 0.000} C_DIS
LIN {X 129.911,Y 216.351,Z 110.000,A 0.000,B 0.000,C 180.000,E1 0.000} C_DIS
LIN {X 118.602,Y 222.751,Z 110.000,A 0.000,B 0.000,C 180.000,E1 0.000} C_DIS
LIN {X 106.978,Y 228.561,Z 110.000,A 0.000,B 0.000,C 180.000,E1 0.000} C_DIS
LIN {X 95.069,Y 233.766,Z 110.000,A 0.000,B 0.000,C 180.000,E1 0.000} C_DIS
LIN {X 82.911,Y 238.349,Z 110.000,A 0.000,B 0.000,C 180.000,E1 0.000} C_DIS
LIN {X 70.530,Y 242.301,Z 110.000,A 0.000,B 0.000,C 180.000,E1 0.000} C_DIS
LIN {X 57.963,Y 245.611,Z 110.000,A 0.000,B 0.000,C 180.000,E1 0.000} C_DIS
LIN {X 45.242,Y 248.269,Z 110.000,A 0.000,B 0.000,C 180.000,E1 0.000} C_DIS
LIN {X 32.403,Y 250.269,Z 110.000,A 0.000,B 0.000,C 180.000,E1 0.000} C_DIS
LIN {X 19.475,Y 251.605,Z 110.000,A 0.000,B 0.000,C 180.000,E1 0.000} C_DIS
LIN {X 6.497,Y 252.274,Z 110.000,A 0.000,B 0.000,C 180.000,E1 0.000} C_DIS
LIN {X -6.497,Y 252.274,Z 110.000,A 0.000,B 0.000,C 180.000,E1 0.000} C_DIS
LIN {X -19.475,Y 251.605,Z 110.000,A 0.000,B 0.000,C 180.000,E1 0.000} C_DIS
LIN {X -32.403,Y 250.269,Z 110.000,A 0.000,B 0.000,C 180.000,E1 0.000} C_DIS
LIN {X -45.242,Y 248.269,Z 110.000,A 0.000,B 0.000,C 180.000,E1 0.000} C_DIS
LIN {X -57.963,Y 245.611,Z 110.000,A 0.000,B 0.000,C 180.000,E1 0.000} C_DIS
LIN {X -70.530,Y 242.301,Z 110.000,A 0.000,B 0.000,C 180.000,E1 0.000} C_DIS
LIN {X -82.910,Y 238.349,Z 110.000,A 0.000,B 0.000,C 180.000,E1 0.000} C_DIS
LIN {X -95.070,Y 233.766,Z 110.000,A 0.000,B 0.000,C 180.000,E1 0.000} C_DIS
LIN {X -106.978,Y 228.561,Z 110.000,A 0.000,B 0.000,C 180.000,E1 0.000} C_DIS
LIN {X -118.602,Y 222.751,Z 110.000,A 0.000,B 0.000,C 180.000,E1 0.000} C_DIS
LIN {X -129.911,Y 216.351,Z 110.000,A 0.000,B 0.000,C 180.000,E1 0.000} C_DIS
LIN {X -140.876,Y 209.375,Z 110.000,A 0.000,B 0.000,C 180.000,E1 0.000} C_DIS
;rapid-leaky
$VEL.CP=0.3
LIN {X 228.114,Y 54.415,Z 110.000,A 0.000,B 0.000,C 180.000,E1 0.000} C_DIS
;bead-sparse_infill
$VEL.CP=0.68
LIN {X 54.327,Y 228.203,Z 110.000,A 0.000,B 0.000,C 180.000,E1 0.000} C_DIS
LIN {X 53.882,Y 228.320,Z 110.000,A 0.000,B 0.000,C 180.000,E1 0.000} C_DIS
LIN {X 42.057,Y 230.791,Z 110.000,A 0.000,B 0.000,C 180.000,E1 0.000} C_DIS
LIN {X 30.122,Y 232.650,Z 110.000,A 0.000,B 0.000,C 180.000,E1 0.000} C_DIS
LIN {X 18.104,Y 233.892,Z 110.000,A 0.000,B 0.000,C 180.000,E1 0.000} C_DIS
LIN {X 6.040,Y 234.514,Z 110.000,A 0.000,B 0.000,C 180.000,E1 0.000} C_DIS
LIN {X -6.040,Y 234.514,Z 110.000,A 0.000,B 0.000,C 180.000,E1 0.000} C_DIS
LIN {X -18.104,Y 233.892,Z 110.000,A 0.000,B 0.000,C 180.000,E1 0.000} C_DIS
LIN {X -30.122,Y 232.650,Z 110.000,A 0.000,B 0.000,C 180.000,E1 0.000} C_DIS
LIN {X -42.057,Y 230.791,Z 110.000,A 0.000,B 0.000,C 180.000,E1 0.000} C_DIS
LIN {X -53.882,Y 228.320,Z 110.000,A 0.000,B 0.000,C 180.000,E1 0.000} C_DIS
LIN {X -65.565,Y 225.243,Z 110.000,A 0.000,B 0.000,C 180.000,E1 0.000} C_DIS
LIN {X -77.074,Y 221.569,Z 110.000,A 0.000,B 0.000,C 180.000,E1 0.000} C_DIS
LIN {X -88.377,Y 217.309,Z 110.000,A 0.000,B 0.000,C 180.000,E1 0.000} C_DIS
LIN {X -90.729,Y 216.281,Z 110.000,A 0.000,B 0.000,C 180.000,E1 0.000} C_DIS
LIN {X 216.271,Y -90.719,Z 110.000,A 0.000,B 0.000,C 180.000,E1 0.000} C_DIS
LIN {X 214.960,Y -93.944,Z 110.000,A 0.000,B 0.000,C 180.000,E1 0.000} C_DIS
LIN {X 209.839,Y -104.886,Z 110.000,A 0.000,B 0.000,C 180.000,E1 0.000} C_DIS
LIN {X 204.163,Y -115.547,Z 110.000,A 0.000,B 0.000,C 180.000,E1 0.000} C_DIS
LIN {X 197.944,Y -125.903,Z 110.000,A 0.000,B 0.000,C 180.000,E1 0.000} C_DIS
LIN {X 191.199,Y -135.927,Z 110.000,A 0.000,B 0.000,C 180.000,E1 0.000} C_DIS
LIN {X 183.947,Y -145.591,Z 110.000,A 0.000,B 0.000,C 180.000,E1 0.000} C_DIS
LIN {X 176.209,Y -154.867,Z 110.000,A 0.000,B 0.000,C 180.000,E1 0.000} C_DIS
LIN {X 168.004,Y -163.731,Z 110.000,A 0.000,B 0.000,C 180.000,E1 0.000} C_DIS
LIN {X 159.353,Y -172.163,Z 110.000,A 0.000,B 0.000,C 180.000,E1 0.000} C_DIS
LIN {X 150.278,Y -180.137,Z 110.000,A 0.000,B 0.000,C 180.000,E1 0.000} C_DIS
LIN {X 149.404,Y -180.829,Z 110.000,A 0.000,B 0.000,C 180.000,E1 0.000} C_DIS
LIN {X -180.795,Y 149.369,Z 110.000,A 0.000,B 0.000,C 180.000,E1 0.000} C_DIS
LIN {X -183.947,Y 145.591,Z 110.000,A 0.000,B 0.000,C 180.000,E1 0.000} C_DIS
LIN {X -191.199,Y 135.927,Z 110.000,A 0.000,B 0.000,C 180.000,E1 0.000} C_DIS
LIN {X -197.944,Y 125.903,Z 110.000,A 0.000,B 0.000,C 180.000,E1 0.000} C_DIS
LIN {X -204.163,Y 115.547,Z 110.000,A 0.000,B 0.000,C 180.000,E1 0.000} C_DIS
LIN {X -209.839,Y 104.886,Z 110.000,A 0.000,B 0.000,C 180.000,E1 0.000} C_DIS
LIN {X -214.960,Y 93.944,Z 110.000,A 0.000,B 0.000,C 180.000,E1 0.000} C_DIS
LIN {X -219.512,Y 82.751,Z 110.000,A 0.000,B 0.000,C 180.000,E1 0.000} C_DIS
LIN {X -223.481,Y 71.343,Z 110.000,A 0.000,B 0.000,C 180.000,E1 0.000} C_DIS
LIN {X -226.856,Y 59.745,Z 110.000,A 0.000,B 0.000,C 180.000,E1 0.000} C_DIS
LIN {X -229.631,Y 47.987,Z 110.000,A 0.000,B 0.000,C 180.000,E1 0.000} C_DIS
LIN {X -230.673,Y 42.269,Z 110.000,A 0.000,B 0.000,C 180.000,E1 0.000} C_DIS
LIN {X 42.330,Y -230.734,Z 110.000,A 0.000,B 0.000,C 180.000,E1 0.000} C_DIS
;rapid-leaky
$VEL.CP=0.3
LIN {X 263.801,Y 0.000,Z 120.000,A 0.000,B 0.000,C 180.000,E1 0.000} C_DIS
;bead-perimeter_outer
$VEL.CP=0.67
LIN {X 263.452,Y 13.580,Z 120.000,A 0.000,B 0.000,C 180.000,E1 0.000} C_DIS
LIN {X 262.403,Y 27.124,Z 120.000,A 0.000,B 0.000,C 180.000,E1 0.000} C_DIS
LIN {X 260.660,Y 40.597,Z 120.000,A 0.000,B 0.000,C 180.000,E1 0.000} C_DIS
LIN {X 258.224,Y 53.961,Z 120.000,A 0.000,B 0.000,C 180.000,E1 0.000} C_DIS
LIN {X 255.103,Y 67.183,Z 120.000,A 0.000,B 0.000,C 180.000,E1 0.000} C_DIS
LIN {X 251.307,Y 80.226,Z 120.000,A 0.000,B 0.000,C 180.000,E1 0.000} C_DIS
LIN {X 246.844,Y 93.056,Z 120.000,A 0.000,B 0.000,C 180.000,E1 0.000} C_DIS
LIN {X 241.726,Y 105.641,Z 120.000,A 0.000,B 0.000,C 180.000,E1 0.000} C_DIS
LIN {X 235.968,Y 117.945,Z 120.000,A 0.000,B 0.000,C 180.000,E1 0.000} C_DIS
LIN {X 229.584,Y 129.934,Z 120.000,A 0.000,B 0.000,C 180.000,E1 0.000} C_DIS
LIN {X 222.589,Y 141.581,Z 120.000,A 0.000,B 0.000,C 180.000,E1 0.000} C_DIS
LIN {X 215.006,Y 152.853,Z 120.000,A 0.000,B 0.000,C 180.000,E1 0.000} C_DIS
LIN {X 206.852,Y 163.718,Z 120.000,A 0.000,B 0.000,C 180.000,E1 0.000} C_DIS
LIN {X 198.151,Y 174.150,Z 120.000,A 0.000,B 0.000,C 180.000,E1 0.000} C_DIS
LIN {X 188.922,Y 184.118,Z 120.000,A 0.000,B 0.000,C 180.000,E1 0.000} C_DIS
LIN {X 179.193,Y 193.600,Z 120.000,A 0.000,B 0.000,C 180.000,E1 0.000} C_DIS
LIN {X 168.989,Y 202.569,Z 120.000,A 0.000,B 0.000,C 180.000,E1 0.000} C_DIS
LIN {X 158.337,Y 211.000,Z 120.000,A 0.000,B 0.000,C 180.000,E1 0.000} C_DIS
LIN {X 147.266,Y 218.870,Z 120.000,A 0.000,B 0.000,C 180.000,E1 0.000} C_DIS
LIN {X 135.804,Y 226.162,Z 120.000,A 0.000,B 0.000,C 180.000,E1 0.000} C_DIS
LIN {X 123.982,Y 232.852,Z 120.000,A 0.000,B 0.000,C 180.000,E1 0.000} C_DIS
LIN {X 111.830,Y 238.926,Z 120.000,A 0.000,B 0.000,C 180.000,E1 0.000} C_DIS
LIN {X 99.381,Y 244.366,Z 120.000,A 0.000,B 0.000,C 180.000,E1 0.000} C_DIS
LIN {X 86.670,Y 249.159,Z 120.000,A 0.000,B 0.000,C 180.000,E1 0.000} C_DIS
LIN {X 73.729,Y 253.289,Z 120.000,A 0.000,B 0.000,C 180.000,E1 0.000} C_DIS
LIN {X 60.591,Y 256.749,Z 120.000,A 0.000,B 0.000,C 180.000,E1 0.000} C_DIS
LIN {X 47.294,Y 259.528,Z 120.000,A 0.000,B 0.000,C 180.000,E1 0.000} C_DIS
LIN {X 33.872,Y 261.618,Z 120.000,A 0.000,B 0.000,C 180.000,E1 0.000} C_DIS
LIN {X 20.359,Y 263.015,Z 120.000,A 0.000,B 0.000,C 180.000,E1 0.000} C_DIS
LIN {X 6.792,Y 263.714,Z 120.000,A 0.000,B 0.000,C 180.000,E1 0.000} C_DIS
LIN {X -6.795,Y 263.714,Z 120.000,A 0.000,B 0.000,C 180.000,E1 0.000} C_DIS
LIN {X -20.359,Y 263.015,Z 120.000,A 0.000,B 0.000,C 180.000,E1 0.000} C_DIS
LIN {X -33.872,Y 261.618,Z 120.000,A 0.000,B 0.000,C 180.000,E1 0.000} C_DIS
LIN {X -47.294,Y 259.528,Z 120.000,A 0.000,B 0.000,C 180.000,E1 0.000} C_DIS
LIN {X -60.591,Y 256.749,Z 120.000,A 0.000,B 0.000,C 180.000,E1 0.000} C_DIS
LIN {X -73.729,Y 253.289,Z 120.000,A 0.000,B 0.000,C 180.000,E1 0.000} C_DIS
LIN {X -86.670,Y 249.159,Z 120.000,A 0.000,B 0.000,C 180.000,E1 0.000} C_DIS
LIN {X -99.381,Y 244.366,Z 120.000,A 0.000,B 0.000,C 180.000,E1 0.000} C_DIS
LIN {X -111.830,Y 238.926,Z 120.000,A 0.000,B 0.000,C 180.000,E1 0.000} C_DIS
LIN {X -123.982,Y 232.852,Z 120.000,A 0.000,B 0.000,C 180.000,E1 0.000} C_DIS
LIN {X -135.804,Y 226.162,Z 120.000,A 0.000,B 0.000,C 180.000,E1 0.000} C_DIS
LIN {X -147.266,Y 218.870,Z 120.000,A 0.000,B 0.000,C 180.000,E1 0.000} C_DIS
LIN {X -158.337,Y 211.000,Z 120.000,A 0.000,B 0.000,C 180.000,E1 0.000} C_DIS
LIN {X -168.989,Y 202.569,Z 120.000,A 0.000,B 0.000,C 180.000,E1 0.000} C_DIS
LIN {X -179.193,Y 193.600,Z 120.000,A 0.000,B 0.000,C 180.000,E1 0.000} C_DIS
LIN {X -188.922,Y 184.118,Z 120.000,A 0.000,B 0.000,C 180.000,E1 0.000} C_DIS
LIN {X -198.151,Y 174.150,Z 120.000,A 0.000,B 0.000,C 180.000,E1 0.000} C_DIS
LIN {X -206.852,Y 163.718,Z 120.000,A 0.000,B 0.000,C 180.000,E1 0.000} C_DIS
LIN {X -215.006,Y 152.853,Z 120.000,A 0.000,B 0.000,C 180.000,E1 0.000} C_DIS
LIN {X -222.589,Y 141.581,Z 120.000,A 0.000,B 0.000,C 180.000,E1 0.000} C_DIS
LIN {X -229.584,Y 129.934,Z 120.000,A 0.000,B 0.000,C 180.000,E1 0.000} C_DIS
LIN {X -235.968,Y 117.945,Z 120.000,A 0.000,B 0.000,C 180.000,E1 0.000} C_DIS
LIN {X -241.726,Y 105.641,Z 120.000,A 0.000,B 0.000,C 180.000,E1 0.000} C_DIS
LIN {X -246.844,Y 93.056,Z 120.000,A 0.000,B 0.000,C 180.000,E1 0.000} C_DIS
LIN {X -251.307,Y 80.226,Z 120.000,A 0.000,B 0.000,C 180.000,E1 0.000} C_DIS
LIN {X -255.103,Y 67.183,Z 120.000,A 0.000,B 0.000,C 180.000,E1 0.000} C_DIS
LIN {X -258.224,Y 53.961,Z 120.000,A 0.000,B 0.000,C 180.000,E1 0.000} C_DIS
LIN {X -260.660,Y 40.597,Z 120.000,A 0.000,B 0.000,C 180.000,E1 0.000} C_DIS
LIN {X -262.403,Y 27.124,Z 120.000,A 0.000,B 0.000,C 180.000,E1 0.000} C_DIS
LIN {X -263.452,Y 13.580,Z 120.000,A 0.000,B 0.000,C 180.000,E1 0.000} C_DIS
LIN {X -263.801,Y 0.000,Z 120.000,A 0.000,B 0.000,C 180.000,E1 0.000} C_DIS
LIN {X -263.452,Y -13.580,Z 120.000,A 0.000,B 0.000,C 180.000,E1 0.000} C_DIS
LIN {X -262.403,Y -27.124,Z 120.000,A 0.000,B 0.000,C 180.000,E1 0.000} C_DIS
LIN {X -260.660,Y -40.597,Z 120.000,A 0.000,B 0.000,C 180.000,E1 0.000} C_DIS
LIN {X -258.224,Y -53.961,Z 120.000,A 0.000,B 0.000,C 180.000,E1 0.000} C_DIS
LIN {X -255.103,Y -67.183,Z 120.000,A 0.000,B 0.000,C 180.000,E1 0.000} C_DIS
LIN {X -251.307,Y -80.226,Z 120.000,A 0.000,B 0.000,C 180.000,E1 0.000} C_DIS
LIN {X -246.844,Y -93.056,Z 120.000,A 0.000,B 0.000,C 180.000,E1 0.000} C_DIS
LIN {X -241.726,Y -105.641,Z 120.000,A 0.000,B 0.000,C 180.000,E1 0.000} C_DIS
LIN {X -235.968,Y -117.945,Z 120.000,A 0.000,B 0.000,C 180.000,E1 0.000} C_DIS
LIN {X -229.584,Y -129.934,Z 120.000,A 0.000,B 0.000,C 180.000,E1 0.000} C_DIS
LIN {X -222.589,Y -141.581,Z 120.000,A 0.000,B 0.000,C 180.000,E1 0.000} C_DIS
LIN {X -215.006,Y -152.853,Z 120.000,A 0.000,B 0.000,C 180.000,E1 0.000} C_DIS
LIN {X -206.852,Y -163.718,Z 120.000,A 0.000,B 0.000,C 180.000,E1 0.000} C_DIS
LIN {X -198.151,Y -174.150,Z 120.000,A 0.000,B 0.000,C 180.000,E1 0.000} C_DIS
LIN {X -188.922,Y -184.118,Z 120.000,A 0.000,B 0.000,C 180.000,E1 0.000} C_DIS
LIN {X -179.193,Y -193.600,Z 120.000,A 0.000,B 0.000,C 180.000,E1 0.000} C_DIS
LIN {X -168.989,Y -202.569,Z 120.000,A 0.000,B 0.000,C 180.000,E1 0.000} C_DIS
LIN {X -158.337,Y -211.000,Z 120.000,A 0.000,B 0.000,C 180.000,E1 0.000} C_DIS
LIN {X -147.266,Y -218.870,Z 120.000,A 0.000,B 0.000,C 180.000,E1 0.000} C_DIS
LIN {X -135.804,Y -226.162,Z 120.000,A 0.000,B 0.000,C 180.000,E1 0.000} C_DIS
LIN {X -123.982,Y -232.852,Z 120.000,A 0.000,B 0.000,C 180.000,E1 0.000} C_DIS
LIN {X -111.830,Y -238.926,Z 120.000,A 0.000,B 0.000,C 180.000,E1 0.000} C_DIS
LIN {X -99.381,Y -244.366,Z 120.000,A 0.000,B 0.000,C 180.000,E1 0.000} C_DIS
LIN {X -86.670,Y -249.159,Z 120.000,A 0.000,B 0.000,C 180.000,E1 0.000} C_DIS
LIN {X -73.729,Y -253.289,Z 120.000,A 0.000,B 0.000,C 180.000,E1 0.000} C_DIS
LIN {X -60.591,Y -256.749,Z 120.000,A 0.000,B 0.000,C 180.000,E1 0.000} C_DIS
LIN {X -47.294,Y -259.528,Z 120.000,A 0.000,B 0.000,C 180.000,E1 0.000} C_DIS
LIN {X -33.872,Y -261.618,Z 120.000,A 0.000,B 0.000,C 180.000,E1 0.000} C_DIS
LIN {X -20.359,Y -263.015,Z 120.000,A 0.000,B 0.000,C 180.000,E1 0.000} C_DIS
LIN {X -6.792,Y -263.714,Z 120.000,A 0.000,B 0.000,C 180.000,E1 0.000} C_DIS
LIN {X 6.795,Y -263.714,Z 120.000,A 0.000,B 0.000,C 180.000,E1 0.000} C_DIS
LIN {X 20.359,Y -263.015,Z 120.000,A 0.000,B 0.000,C 180.000,E1 0.000} C_DIS
LIN {X 33.872,Y -261.618,Z 120.000,A 0.000,B 0.000,C 180.000,E1 0.000} C_DIS
LIN {X 47.294,Y -259.528,Z 120.000,A 0.000,B 0.000,C 180.000,E1 0.000} C_DIS
LIN {X 60.591,Y -256.749,Z 120.000,A 0.000,B 0.000,C 180.000,E1 0.000} C_DIS
LIN {X 73.729,Y -253.289,Z 120.000,A 0.000,B 0.000,C 180.000,E1 0.000} C_DIS
LIN {X 86.670,Y -249.159,Z 120.000,A 0.000,B 0.000,C 180.000,E1 0.000} C_DIS
LIN {X 99.381,Y -244.366,Z 120.000,A 0.000,B 0.000,C 180.000,E1 0.000} C_DIS
LIN {X 111.830,Y -238.926,Z 120.000,A 0.000,B 0.000,C 180.000,E1 0.000} C_DIS
LIN {X 123.982,Y -232.852,Z 120.000,A 0.000,B 0.000,C 180.000,E1 0.000} C_DIS
LIN {X 135.804,Y -226.162,Z 120.000,A 0.000,B 0.000,C 180.000,E1 0.000} C_DIS
LIN {X 147.266,Y -218.870,Z 120.000,A 0.000,B 0.000,C 180.000,E1 0.000} C_DIS
LIN {X 158.337,Y -211.000,Z 120.000,A 0.000,B 0.000,C 180.000,E1 0.000} C_DIS
LIN {X 168.989,Y -202.569,Z 120.000,A 0.000,B 0.000,C 180.000,E1 0.000} C_DIS
LIN {X 179.193,Y -193.600,Z 120.000,A 0.000,B 0.000,C 180.000,E1 0.000} C_DIS
LIN {X 188.922,Y -184.118,Z 120.000,A 0.000,B 0.000,C 180.000,E1 0.000} C_DIS
LIN {X 198.151,Y -174.150,Z 120.000,A 0.000,B 0.000,C 180.000,E1 0.000} C_DIS
LIN {X 206.852,Y -163.718,Z 120.000,A 0.000,B 0.000,C 180.000,E1 0.000} C_DIS
LIN {X 215.006,Y -152.853,Z 120.000,A 0.000,B 0.000,C 180.000,E1 0.000} C_DIS
LIN {X 222.589,Y -141.581,Z 120.000,A 0.000,B 0.000,C 180.000,E1 0.000} C_DIS
LIN {X 229.584,Y -129.934,Z 120.000,A 0.000,B 0.000,C 180.000,E1 0.000} C_DIS
LIN {X 235.968,Y -117.945,Z 120.000,A 0.000,B 0.000,C 180.000,E1 0.000} C_DIS
LIN {X 241.726,Y -105.641,Z 120.000,A 0.000,B 0.000,C 180.000,E1 0.000} C_DIS
LIN {X 246.844,Y -93.056,Z 120.000,A 0.000,B 0.000,C 180.000,E1 0.000} C_DIS
LIN {X 251.307,Y -80.226,Z 120.000,A 0.000,B 0.000,C 180.000,E1 0.000} C_DIS
LIN {X 255.103,Y -67.183,Z 120.000,A 0.000,B 0.000,C 180.000,E1 0.000} C_DIS
LIN {X 258.224,Y -53.961,Z 120.000,A 0.000,B 0.000,C 180.000,E1 0.000} C_DIS
LIN {X 260.660,Y -40.597,Z 120.000,A 0.000,B 0.000,C 180.000,E1 0.000} C_DIS
LIN {X 262.403,Y -27.124,Z 120.000,A 0.000,B 0.000,C 180.000,E1 0.000} C_DIS
LIN {X 263.452,Y -13.580,Z 120.000,A 0.000,B 0.000,C 180.000,E1 0.000} C_DIS
LIN {X 263.801,Y 0.000,Z 120.000,A 0.000,B 0.000,C 180.000,E1 0.000} C_DIS
;rapid-leaky
$VEL.CP=0.3
LIN {X 248.256,Y 0.000,Z 120.000,A 0.000,B 0.000,C 180.000,E1 0.000} C_DIS
;bead-perimeter_inner
$VEL.CP=0.67
LIN {X 247.927,Y 12.780,Z 120.000,A 0.000,B 0.000,C 180.000,E1 0.000} C_DIS
LIN {X 246.940,Y 25.526,Z 120.000,A 0.000,B 0.000,C 180.000,E1 0.000} C_DIS
LIN {X 245.300,Y 38.205,Z 120.000,A 0.000,B 0.000,C 180.000,E1 0.000} C_DIS
LIN {X 243.008,Y 50.781,Z 120.000,A 0.000,B 0.000,C 180.000,E1 0.000} C_DIS
LIN {X 240.071,Y 63.225,Z 120.000,A 0.000,B 0.000,C 180.000,E1 0.000} C_DIS
LIN {X 236.498,Y 75.499,Z 120.000,A 0.000,B 0.000,C 180.000,E1 0.000} C_DIS
LIN {X 232.298,Y 87.573,Z 120.000,A 0.000,B 0.000,C 180.000,E1 0.000} C_DIS
LIN {X 227.482,Y 99.416,Z 120.000,A 0.000,B 0.000,C 180.000,E1 0.000} C_DIS
LIN {X 222.063,Y 110.995,Z 120.000,A 0.000,B 0.000,C 180.000,E1 0.000} C_DIS
LIN {X 216.056,Y 122.277,Z 120.000,A 0.000,B 0.000,C 180.000,E1 0.000} C_DIS
LIN {X 209.473,Y 133.237,Z 120.000,A 0.000,B 0.000,C 180.000,E1 0.000} C_DIS
LIN {X 202.336,Y 143.846,Z 120.000,A 0.000,B 0.000,C 180.000,E1 0.000} C_DIS
LIN {X 194.663,Y 154.071,Z 120.000,A 0.000,B 0.000,C 180.000,E1 0.000} C_DIS
LIN {X 186.475,Y 163.887,Z 120.000,A 0.000,B 0.000,C 180.000,E1 0.000} C_DIS
LIN {X 177.790,Y 173.268,Z 120.000,A 0.000,B 0.000,C 180.000,E1 0.000} C_DIS
LIN {X 168.634,Y 182.192,Z 120.000,A 0.000,B 0.000,C 180.000,E1 0.000} C_DIS
LIN {X 159.031,Y 190.632,Z 120.000,A 0.000,B 0.000,C 180.000,E1 0.000} C_DIS
LIN {X 149.007,Y 198.566,Z 120.000,A 0.000,B 0.000,C 180.000,E1 0.000} C_DIS
LIN {X 138.588,Y 205.972,Z 120.000,A 0.000,B 0.000,C 180.000,E1 0.000} C_DIS
LIN {X 127.801,Y 212.835,Z 120.000,A 0.000,B 0.000,C 180.000,E1 0.000} C_DIS
LIN {X 116.676,Y 219.131,Z 120.000,A 0.000,B 0.000,C 180.000,E1 0.000} C_DIS
LIN {X 105.240,Y 224.847,Z 120.000,A 0.000,B 0.000,C 180.000,E1 0.000} C_DIS
LIN {X 93.525,Y 229.967,Z 120.000,A 0.000,B 0.000,C 180.000,E1 0.000} C_DIS
LIN {X 81.563,Y 234.476,Z 120.000,A 0.000,B 0.000,C 180.000,E1 0.000} C_DIS
LIN {X 69.385,Y 238.363,Z 120.000,A 0.000,B 0.000,C 180.000,E1 0.000} C_DIS
LIN {X 57.020,Y 241.620,Z 120.000,A 0.000,B 0.000,C 180.000,E1 0.000} C_DIS
LIN {X 44.507,Y 244.235,Z 120.000,A 0.000,B 0.000,C 180.000,E1 0.000} C_DIS
LIN {X 31.876,Y 246.202,Z 120.000,A 0.000,B 0.000,C 180.000,E1 0.000} C_DIS
LIN {X 19.160,Y 247.517,Z 120.000,A 0.000,B 0.000,C 180.000,E1 0.000} C_DIS
LIN {X 6.393,Y 248.174,Z 120.000,A 0.000,B 0.000,C 180.000,E1 0.000} C_DIS
